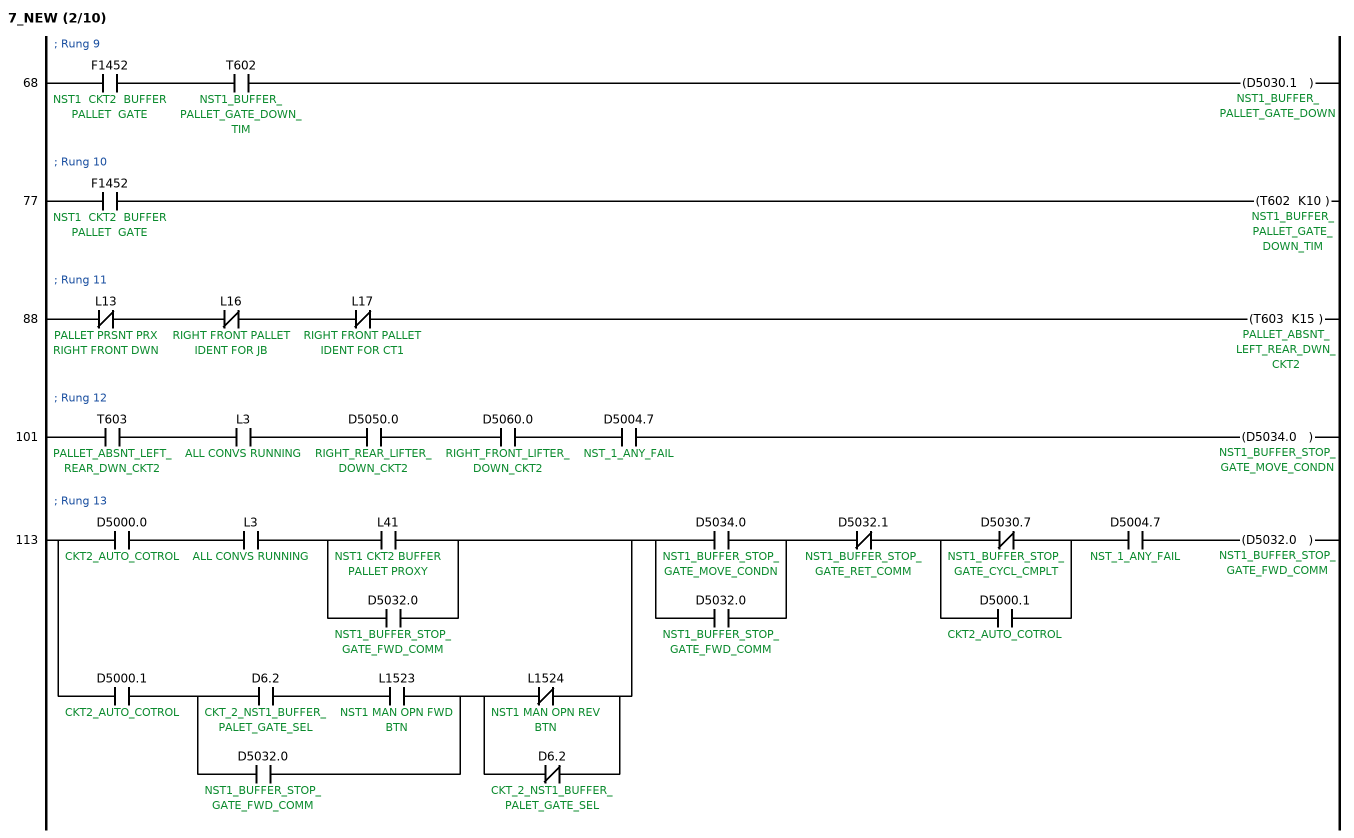
[picture p72: ladder of 7_NEW, rungs at steps 68 to 113]
; Rung 9
68    LD      F1452  ; NST1  CKT2  BUFFER  PALLET  GATE
      AND     T602  ; NST1_BUFFER_PALLET_GATE_DOWN_TIM
      OUT     D5030.1  ; NST1_BUFFER_PALLET_GATE_DOWN
; Rung 10
77    LD      F1452  ; NST1  CKT2  BUFFER  PALLET  GATE
      OUT     T602 K10  ; NST1_BUFFER_PALLET_GATE_DOWN_TIM
; Rung 11
88    LDI     L13  ; PALLET PRSNT PRX RIGHT FRONT DWN
      ANI     L16  ; RIGHT FRONT PALLET IDENT FOR JB
      ANI     L17  ; RIGHT FRONT PALLET IDENT FOR CT1
      OUT     T603 K15  ; PALLET_ABSNT_LEFT_REAR_DWN_CKT2
; Rung 12
101   LD      T603  ; PALLET_ABSNT_LEFT_REAR_DWN_CKT2
      AND     L3  ; ALL CONVS RUNNING
      AND     D5050.0  ; RIGHT_REAR_LIFTER_DOWN_CKT2
      AND     D5060.0  ; RIGHT_FRONT_LIFTER_DOWN_CKT2
      AND     D5004.7  ; NST_1_ANY_FAIL
      OUT     D5034.0  ; NST1_BUFFER_STOP_GATE_MOVE_CONDN
; Rung 13
113   LD      D5000.0  ; CKT2_AUTO_COTROL
      AND     L3  ; ALL CONVS RUNNING
      LD      L41  ; NST1 CKT2 BUFFER PALLET PROXY
      OR      D5032.0  ; NST1_BUFFER_STOP_GATE_FWD_COMM
      ANB
      LD      D5000.1  ; CKT2_AUTO_COTROL
      LD      D6.2  ; CKT_2_NST1_BUFFER_PALET_GATE_SEL
      AND     L1523  ; NST1 MAN OPN FWD BTN
      OR      D5032.0  ; NST1_BUFFER_STOP_GATE_FWD_COMM
      ANB
      LDI     L1524  ; NST1 MAN OPN REV BTN
      ORI     D6.2  ; CKT_2_NST1_BUFFER_PALET_GATE_SEL
      ANB
      ORB
      LD      D5034.0  ; NST1_BUFFER_STOP_GATE_MOVE_CONDN
      OR      D5032.0  ; NST1_BUFFER_STOP_GATE_FWD_COMM
      ANB
      ANI     D5032.1  ; NST1_BUFFER_STOP_GATE_RET_COMM
      LDI     D5030.7  ; NST1_BUFFER_STOP_GATE_CYCL_CMPLT
      OR      D5000.1  ; CKT2_AUTO_COTROL
      ANB
      AND     D5004.7  ; NST_1_ANY_FAIL
      OUT     D5032.0  ; NST1_BUFFER_STOP_GATE_FWD_COMM
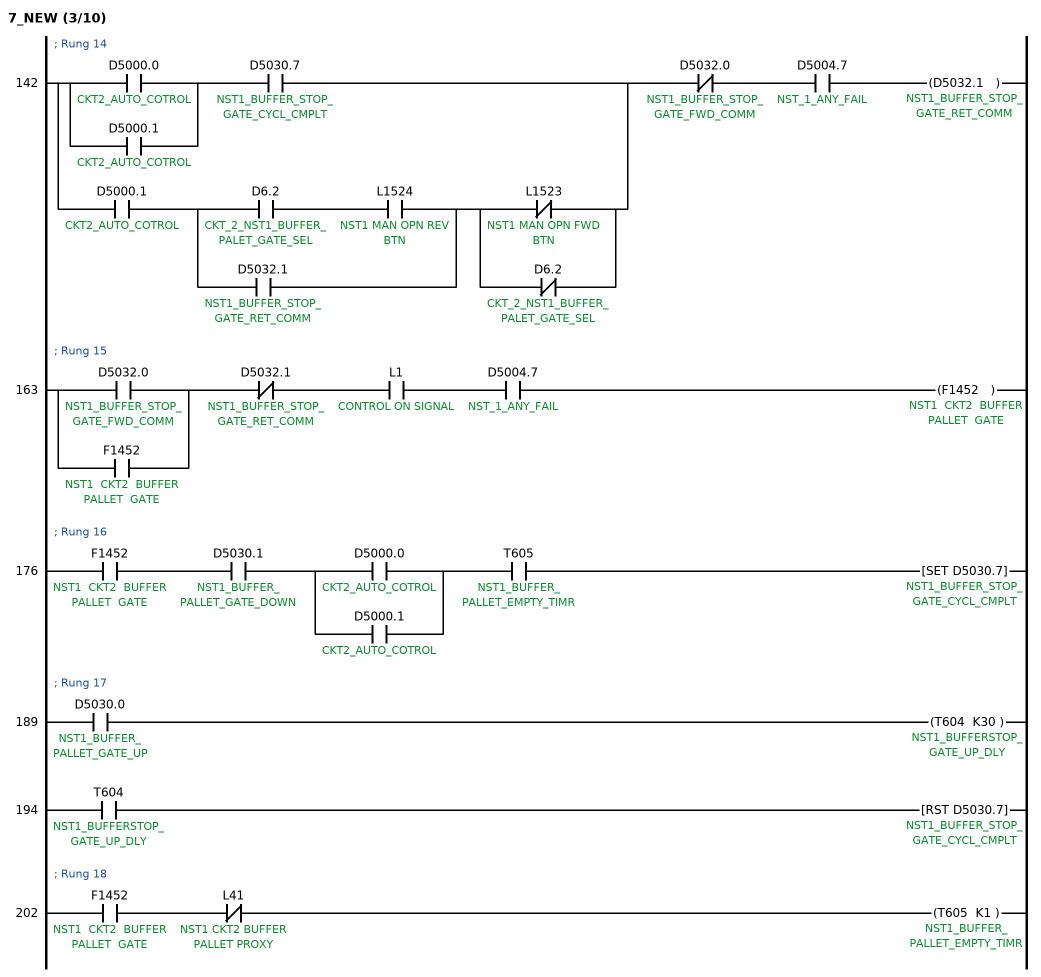
; Rung 14
142   LD      D5000.0  ; CKT2_AUTO_COTROL
      OR      D5000.1  ; CKT2_AUTO_COTROL
      AND     D5030.7  ; NST1_BUFFER_STOP_GATE_CYCL_CMPLT
      LD      D5000.1  ; CKT2_AUTO_COTROL
      LD      D6.2  ; CKT_2_NST1_BUFFER_PALET_GATE_SEL
      AND     L1524  ; NST1 MAN OPN REV BTN
      OR      D5032.1  ; NST1_BUFFER_STOP_GATE_RET_COMM
      ANB
      LDI     L1523  ; NST1 MAN OPN FWD BTN
      ORI     D6.2  ; CKT_2_NST1_BUFFER_PALET_GATE_SEL
      ANB
      ORB
      ANI     D5032.0  ; NST1_BUFFER_STOP_GATE_FWD_COMM
      AND     D5004.7  ; NST_1_ANY_FAIL
      OUT     D5032.1  ; NST1_BUFFER_STOP_GATE_RET_COMM
; Rung 15
163   LD      D5032.0  ; NST1_BUFFER_STOP_GATE_FWD_COMM
      OR      F1452  ; NST1  CKT2  BUFFER  PALLET  GATE
      ANI     D5032.1  ; NST1_BUFFER_STOP_GATE_RET_COMM
      AND     L1  ; CONTROL ON SIGNAL
      AND     D5004.7  ; NST_1_ANY_FAIL
      OUT     F1452  ; NST1  CKT2  BUFFER  PALLET  GATE
; Rung 16
176   LD      F1452  ; NST1  CKT2  BUFFER  PALLET  GATE
      AND     D5030.1  ; NST1_BUFFER_PALLET_GATE_DOWN
      LD      D5000.0  ; CKT2_AUTO_COTROL
      OR      D5000.1  ; CKT2_AUTO_COTROL
      ANB
      AND     T605  ; NST1_BUFFER_PALLET_EMPTY_TIMR
      SET     D5030.7  ; NST1_BUFFER_STOP_GATE_CYCL_CMPLT
; Rung 17
189   LD      D5030.0  ; NST1_BUFFER_PALLET_GATE_UP
      OUT     T604 K30  ; NST1_BUFFERSTOP_GATE_UP_DLY
194   LD      T604  ; NST1_BUFFERSTOP_GATE_UP_DLY
      RST     D5030.7  ; NST1_BUFFER_STOP_GATE_CYCL_CMPLT
; Rung 18
202   LD      F1452  ; NST1  CKT2  BUFFER  PALLET  GATE
      ANI     L41  ; NST1 CKT2 BUFFER PALLET PROXY
      OUT     T605 K1  ; NST1_BUFFER_PALLET_EMPTY_TIMR
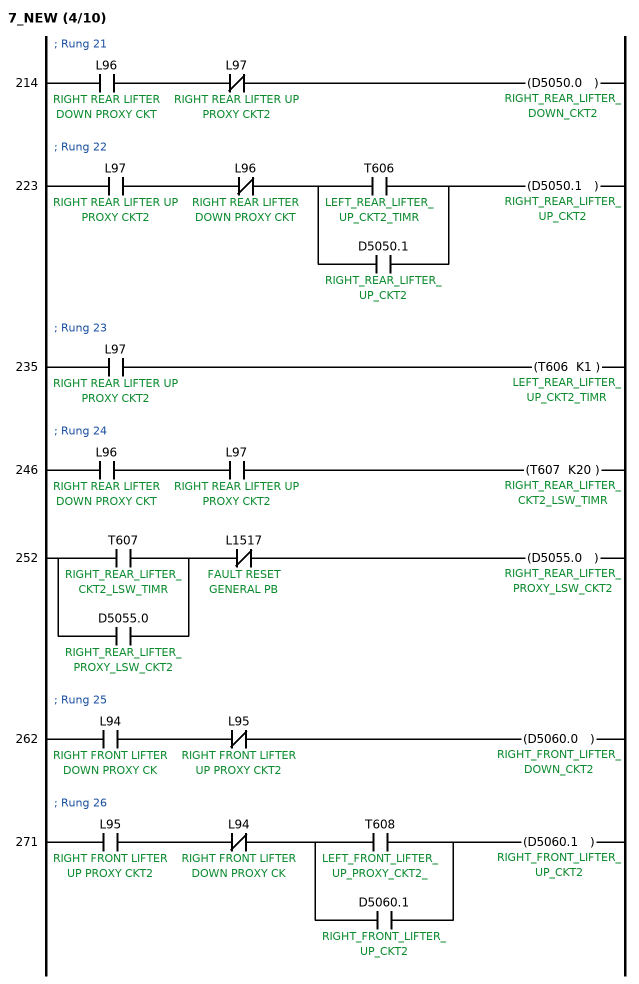
; Rung 21
214   LD      L96  ; RIGHT REAR LIFTER DOWN PROXY CKT
      ANI     L97  ; RIGHT REAR LIFTER UP PROXY CKT2
      OUT     D5050.0  ; RIGHT_REAR_LIFTER_DOWN_CKT2
; Rung 22
223   LD      L97  ; RIGHT REAR LIFTER UP PROXY CKT2
      ANI     L96  ; RIGHT REAR LIFTER DOWN PROXY CKT
      LD      T606  ; LEFT_REAR_LIFTER_UP_CKT2_TIMR
      OR      D5050.1  ; RIGHT_REAR_LIFTER_UP_CKT2
      ANB
      OUT     D5050.1  ; RIGHT_REAR_LIFTER_UP_CKT2
; Rung 23
235   LD      L97  ; RIGHT REAR LIFTER UP PROXY CKT2
      OUT     T606 K1  ; LEFT_REAR_LIFTER_UP_CKT2_TIMR
; Rung 24
246   LD      L96  ; RIGHT REAR LIFTER DOWN PROXY CKT
      AND     L97  ; RIGHT REAR LIFTER UP PROXY CKT2
      OUT     T607 K20  ; RIGHT_REAR_LIFTER_CKT2_LSW_TIMR
252   LD      T607  ; RIGHT_REAR_LIFTER_CKT2_LSW_TIMR
      OR      D5055.0  ; RIGHT_REAR_LIFTER_PROXY_LSW_CKT2
      ANI     L1517  ; FAULT RESET GENERAL PB
      OUT     D5055.0  ; RIGHT_REAR_LIFTER_PROXY_LSW_CKT2
; Rung 25
262   LD      L94  ; RIGHT FRONT LIFTER DOWN PROXY CK
      ANI     L95  ; RIGHT FRONT LIFTER UP PROXY CKT2
      OUT     D5060.0  ; RIGHT_FRONT_LIFTER_DOWN_CKT2
; Rung 26
271   LD      L95  ; RIGHT FRONT LIFTER UP PROXY CKT2
      ANI     L94  ; RIGHT FRONT LIFTER DOWN PROXY CK
      LD      T608  ; LEFT_FRONT_LIFTER_UP_PROXY_CKT2_
      OR      D5060.1  ; RIGHT_FRONT_LIFTER_UP_CKT2
      ANB
      OUT     D5060.1  ; RIGHT_FRONT_LIFTER_UP_CKT2
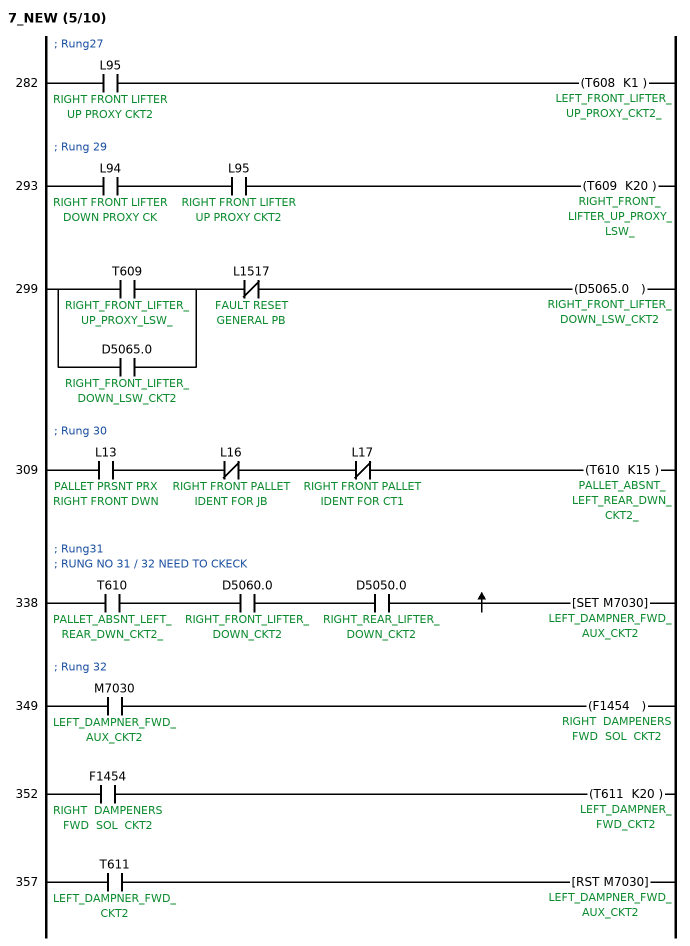
; Rung27
282   LD      L95  ; RIGHT FRONT LIFTER UP PROXY CKT2
      OUT     T608 K1  ; LEFT_FRONT_LIFTER_UP_PROXY_CKT2_
; Rung 29
293   LD      L94  ; RIGHT FRONT LIFTER DOWN PROXY CK
      AND     L95  ; RIGHT FRONT LIFTER UP PROXY CKT2
      OUT     T609 K20  ; RIGHT_FRONT_LIFTER_UP_PROXY_LSW_
299   LD      T609  ; RIGHT_FRONT_LIFTER_UP_PROXY_LSW_
      OR      D5065.0  ; RIGHT_FRONT_LIFTER_DOWN_LSW_CKT2
      ANI     L1517  ; FAULT RESET GENERAL PB
      OUT     D5065.0  ; RIGHT_FRONT_LIFTER_DOWN_LSW_CKT2
; Rung 30
309   LD      L13  ; PALLET PRSNT PRX RIGHT FRONT DWN
      ANI     L16  ; RIGHT FRONT PALLET IDENT FOR JB
      ANI     L17  ; RIGHT FRONT PALLET IDENT FOR CT1
      OUT     T610 K15  ; PALLET_ABSNT_LEFT_REAR_DWN_CKT2_
; Rung31
; RUNG NO 31 / 32 NEED TO CKECK
338   LD      T610  ; PALLET_ABSNT_LEFT_REAR_DWN_CKT2_
      AND     D5060.0  ; RIGHT_FRONT_LIFTER_DOWN_CKT2
      AND     D5050.0  ; RIGHT_REAR_LIFTER_DOWN_CKT2
      MEP
      SET     M7030  ; LEFT_DAMPNER_FWD_AUX_CKT2
; Rung 32
349   LD      M7030  ; LEFT_DAMPNER_FWD_AUX_CKT2
      OUT     F1454  ; RIGHT  DAMPENERS  FWD  SOL  CKT2
352   LD      F1454  ; RIGHT  DAMPENERS  FWD  SOL  CKT2
      OUT     T611 K20  ; LEFT_DAMPNER_FWD_CKT2
357   LD      T611  ; LEFT_DAMPNER_FWD_CKT2
      RST     M7030  ; LEFT_DAMPNER_FWD_AUX_CKT2
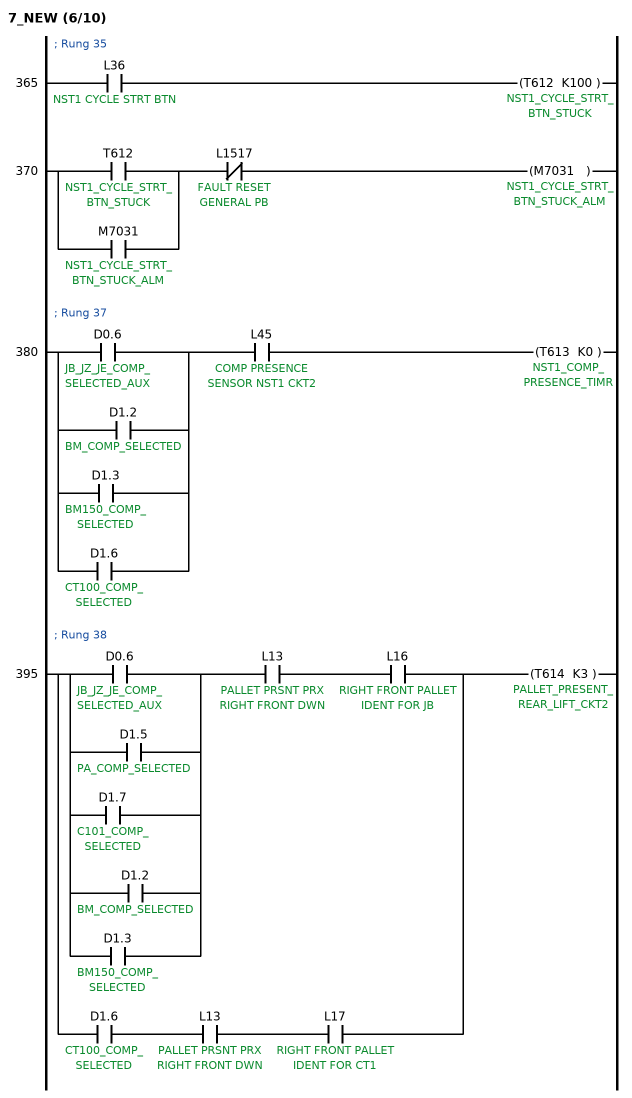
; Rung 35
365   LD      L36  ; NST1 CYCLE STRT BTN
      OUT     T612 K100  ; NST1_CYCLE_STRT_BTN_STUCK
370   LD      T612  ; NST1_CYCLE_STRT_BTN_STUCK
      OR      M7031  ; NST1_CYCLE_STRT_BTN_STUCK_ALM
      ANI     L1517  ; FAULT RESET GENERAL PB
      OUT     M7031  ; NST1_CYCLE_STRT_BTN_STUCK_ALM
; Rung 37
380   LD      D0.6  ; JB_JZ_JE_COMP_SELECTED_AUX
      OR      D1.2  ; BM_COMP_SELECTED
      OR      D1.3  ; BM150_COMP_SELECTED
      OR      D1.6  ; CT100_COMP_SELECTED
      AND     L45  ; COMP PRESENCE SENSOR NST1 CKT2
      OUT     T613 K0  ; NST1_COMP_PRESENCE_TIMR
; Rung 38
395   LD      D0.6  ; JB_JZ_JE_COMP_SELECTED_AUX
      OR      D1.5  ; PA_COMP_SELECTED
      OR      D1.7  ; C101_COMP_SELECTED
      OR      D1.2  ; BM_COMP_SELECTED
      OR      D1.3  ; BM150_COMP_SELECTED
      AND     L13  ; PALLET PRSNT PRX RIGHT FRONT DWN
      AND     L16  ; RIGHT FRONT PALLET IDENT FOR JB
      LD      D1.6  ; CT100_COMP_SELECTED
      AND     L13  ; PALLET PRSNT PRX RIGHT FRONT DWN
      AND     L17  ; RIGHT FRONT PALLET IDENT FOR CT1
      ORB
      OUT     T614 K3  ; PALLET_PRESENT_REAR_LIFT_CKT2
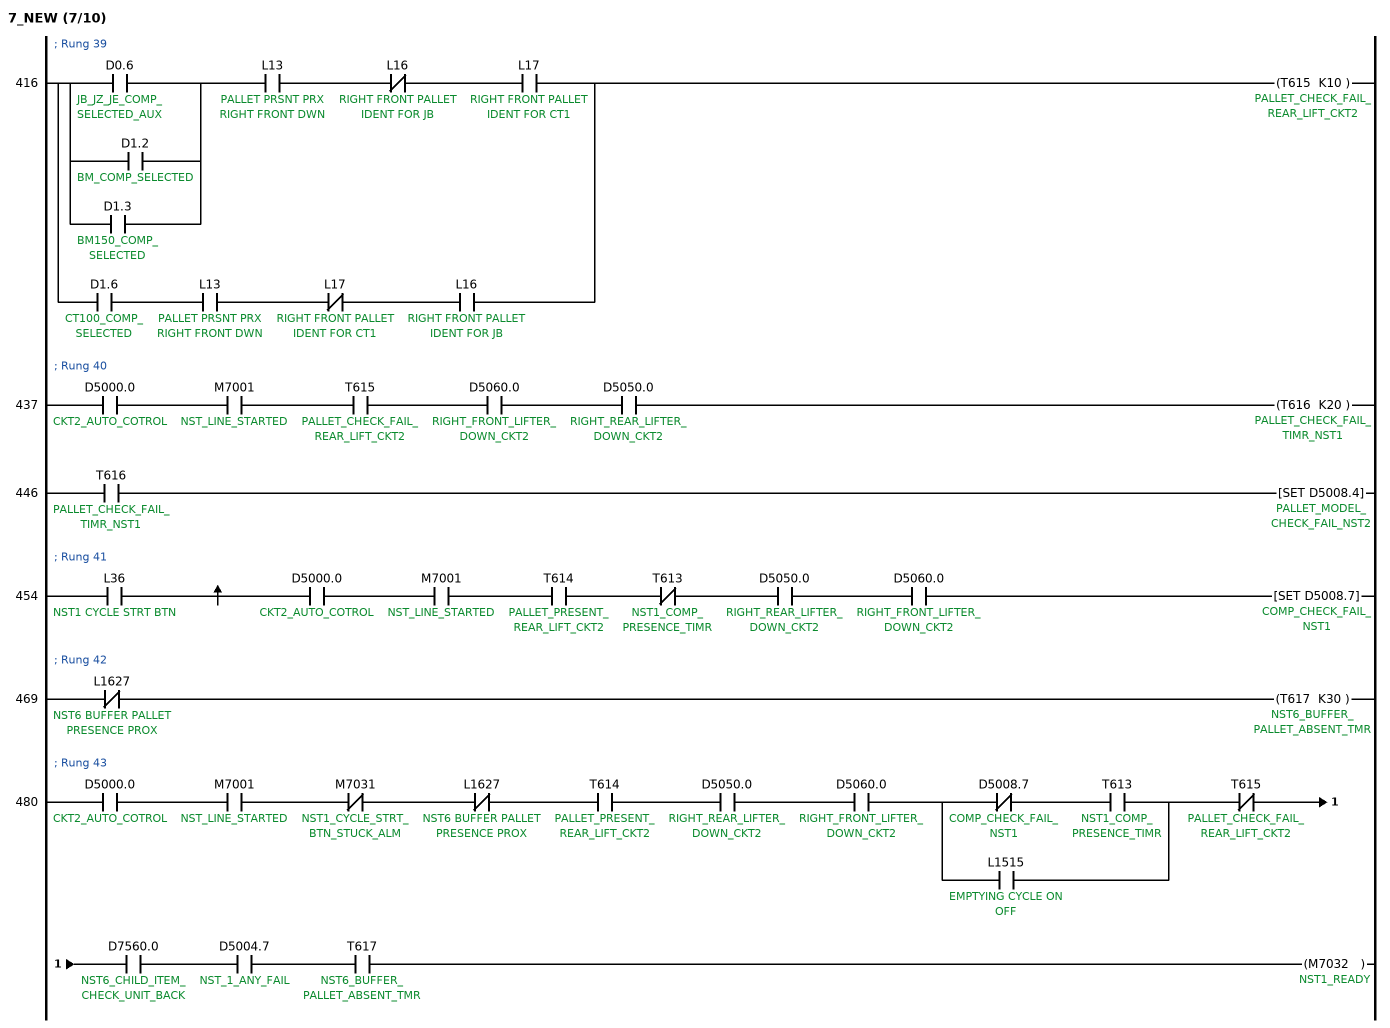
; Rung 39
416   LD      D0.6  ; JB_JZ_JE_COMP_SELECTED_AUX
      OR      D1.2  ; BM_COMP_SELECTED
      OR      D1.3  ; BM150_COMP_SELECTED
      AND     L13  ; PALLET PRSNT PRX RIGHT FRONT DWN
      ANI     L16  ; RIGHT FRONT PALLET IDENT FOR JB
      AND     L17  ; RIGHT FRONT PALLET IDENT FOR CT1
      LD      D1.6  ; CT100_COMP_SELECTED
      AND     L13  ; PALLET PRSNT PRX RIGHT FRONT DWN
      ANI     L17  ; RIGHT FRONT PALLET IDENT FOR CT1
      AND     L16  ; RIGHT FRONT PALLET IDENT FOR JB
      ORB
      OUT     T615 K10  ; PALLET_CHECK_FAIL_REAR_LIFT_CKT2
; Rung 40
437   LD      D5000.0  ; CKT2_AUTO_COTROL
      AND     M7001  ; NST_LINE_STARTED
      AND     T615  ; PALLET_CHECK_FAIL_REAR_LIFT_CKT2
      AND     D5060.0  ; RIGHT_FRONT_LIFTER_DOWN_CKT2
      AND     D5050.0  ; RIGHT_REAR_LIFTER_DOWN_CKT2
      OUT     T616 K20  ; PALLET_CHECK_FAIL_TIMR_NST1
446   LD      T616  ; PALLET_CHECK_FAIL_TIMR_NST1
      SET     D5008.4  ; PALLET_MODEL_CHECK_FAIL_NST2
; Rung 41
454   LD      L36  ; NST1 CYCLE STRT BTN
      MEP
      AND     D5000.0  ; CKT2_AUTO_COTROL
      AND     M7001  ; NST_LINE_STARTED
      AND     T614  ; PALLET_PRESENT_REAR_LIFT_CKT2
      ANI     T613  ; NST1_COMP_PRESENCE_TIMR
      AND     D5050.0  ; RIGHT_REAR_LIFTER_DOWN_CKT2
      AND     D5060.0  ; RIGHT_FRONT_LIFTER_DOWN_CKT2
      SET     D5008.7  ; COMP_CHECK_FAIL_NST1
; Rung 42
469   LDI     L1627  ; NST6 BUFFER PALLET PRESENCE PROX
      OUT     T617 K30  ; NST6_BUFFER_PALLET_ABSENT_TMR
; Rung 43
480   LD      D5000.0  ; CKT2_AUTO_COTROL
      AND     M7001  ; NST_LINE_STARTED
      ANI     M7031  ; NST1_CYCLE_STRT_BTN_STUCK_ALM
      ANI     L1627  ; NST6 BUFFER PALLET PRESENCE PROX
      AND     T614  ; PALLET_PRESENT_REAR_LIFT_CKT2
      AND     D5050.0  ; RIGHT_REAR_LIFTER_DOWN_CKT2
      AND     D5060.0  ; RIGHT_FRONT_LIFTER_DOWN_CKT2
      LDI     D5008.7  ; COMP_CHECK_FAIL_NST1
      AND     T613  ; NST1_COMP_PRESENCE_TIMR
      OR      L1515  ; EMPTYING CYCLE ON OFF
      ANB
      ANI     T615  ; PALLET_CHECK_FAIL_REAR_LIFT_CKT2
      AND     D7560.0  ; NST6_CHILD_ITEM_CHECK_UNIT_BACK
      AND     D5004.7  ; NST_1_ANY_FAIL
      AND     T617  ; NST6_BUFFER_PALLET_ABSENT_TMR
      OUT     M7032  ; NST1_READY
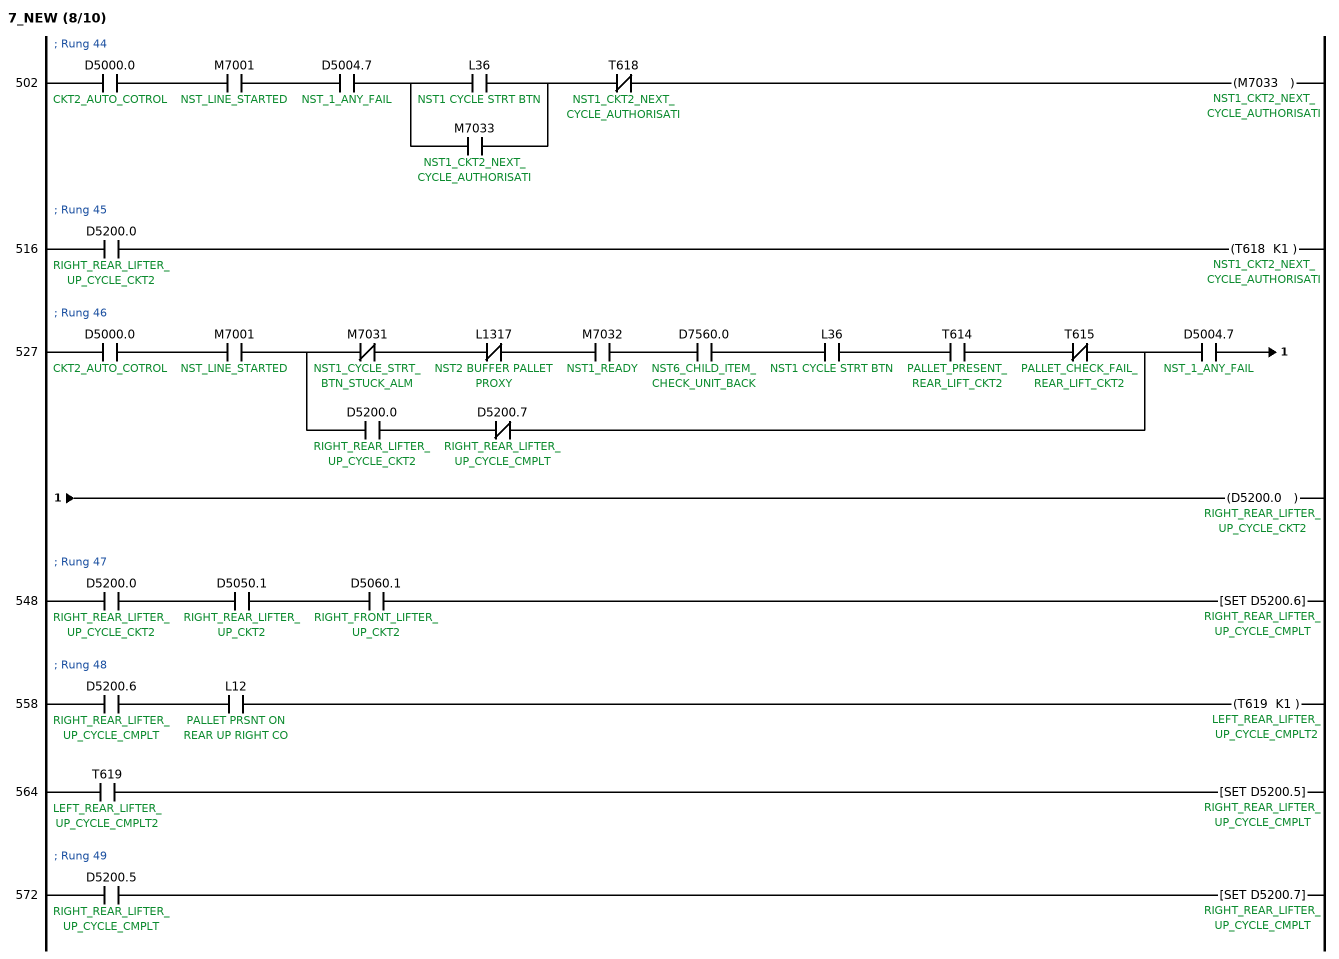
; Rung 44
502   LD      D5000.0  ; CKT2_AUTO_COTROL
      AND     M7001  ; NST_LINE_STARTED
      AND     D5004.7  ; NST_1_ANY_FAIL
      LD      L36  ; NST1 CYCLE STRT BTN
      OR      M7033  ; NST1_CKT2_NEXT_CYCLE_AUTHORISATI
      ANB
      ANI     T618  ; NST1_CKT2_NEXT_CYCLE_AUTHORISATI
      OUT     M7033  ; NST1_CKT2_NEXT_CYCLE_AUTHORISATI
; Rung 45
516   LD      D5200.0  ; RIGHT_REAR_LIFTER_UP_CYCLE_CKT2
      OUT     T618 K1  ; NST1_CKT2_NEXT_CYCLE_AUTHORISATI
; Rung 46
527   LD      D5000.0  ; CKT2_AUTO_COTROL
      AND     M7001  ; NST_LINE_STARTED
      LDI     M7031  ; NST1_CYCLE_STRT_BTN_STUCK_ALM
      ANI     L1317  ; NST2 BUFFER PALLET PROXY
      AND     M7032  ; NST1_READY
      AND     D7560.0  ; NST6_CHILD_ITEM_CHECK_UNIT_BACK
      AND     L36  ; NST1 CYCLE STRT BTN
      AND     T614  ; PALLET_PRESENT_REAR_LIFT_CKT2
      ANI     T615  ; PALLET_CHECK_FAIL_REAR_LIFT_CKT2
      LD      D5200.0  ; RIGHT_REAR_LIFTER_UP_CYCLE_CKT2
      ANI     D5200.7  ; RIGHT_REAR_LIFTER_UP_CYCLE_CMPLT
      ORB
      ANB
      AND     D5004.7  ; NST_1_ANY_FAIL
      OUT     D5200.0  ; RIGHT_REAR_LIFTER_UP_CYCLE_CKT2
; Rung 47
548   LD      D5200.0  ; RIGHT_REAR_LIFTER_UP_CYCLE_CKT2
      AND     D5050.1  ; RIGHT_REAR_LIFTER_UP_CKT2
      AND     D5060.1  ; RIGHT_FRONT_LIFTER_UP_CKT2
      SET     D5200.6  ; RIGHT_REAR_LIFTER_UP_CYCLE_CMPLT
; Rung 48
558   LD      D5200.6  ; RIGHT_REAR_LIFTER_UP_CYCLE_CMPLT
      AND     L12  ; PALLET PRSNT ON REAR UP RIGHT CO
      OUT     T619 K1  ; LEFT_REAR_LIFTER_UP_CYCLE_CMPLT2
564   LD      T619  ; LEFT_REAR_LIFTER_UP_CYCLE_CMPLT2
      SET     D5200.5  ; RIGHT_REAR_LIFTER_UP_CYCLE_CMPLT
; Rung 49
572   LD      D5200.5  ; RIGHT_REAR_LIFTER_UP_CYCLE_CMPLT
      SET     D5200.7  ; RIGHT_REAR_LIFTER_UP_CYCLE_CMPLT
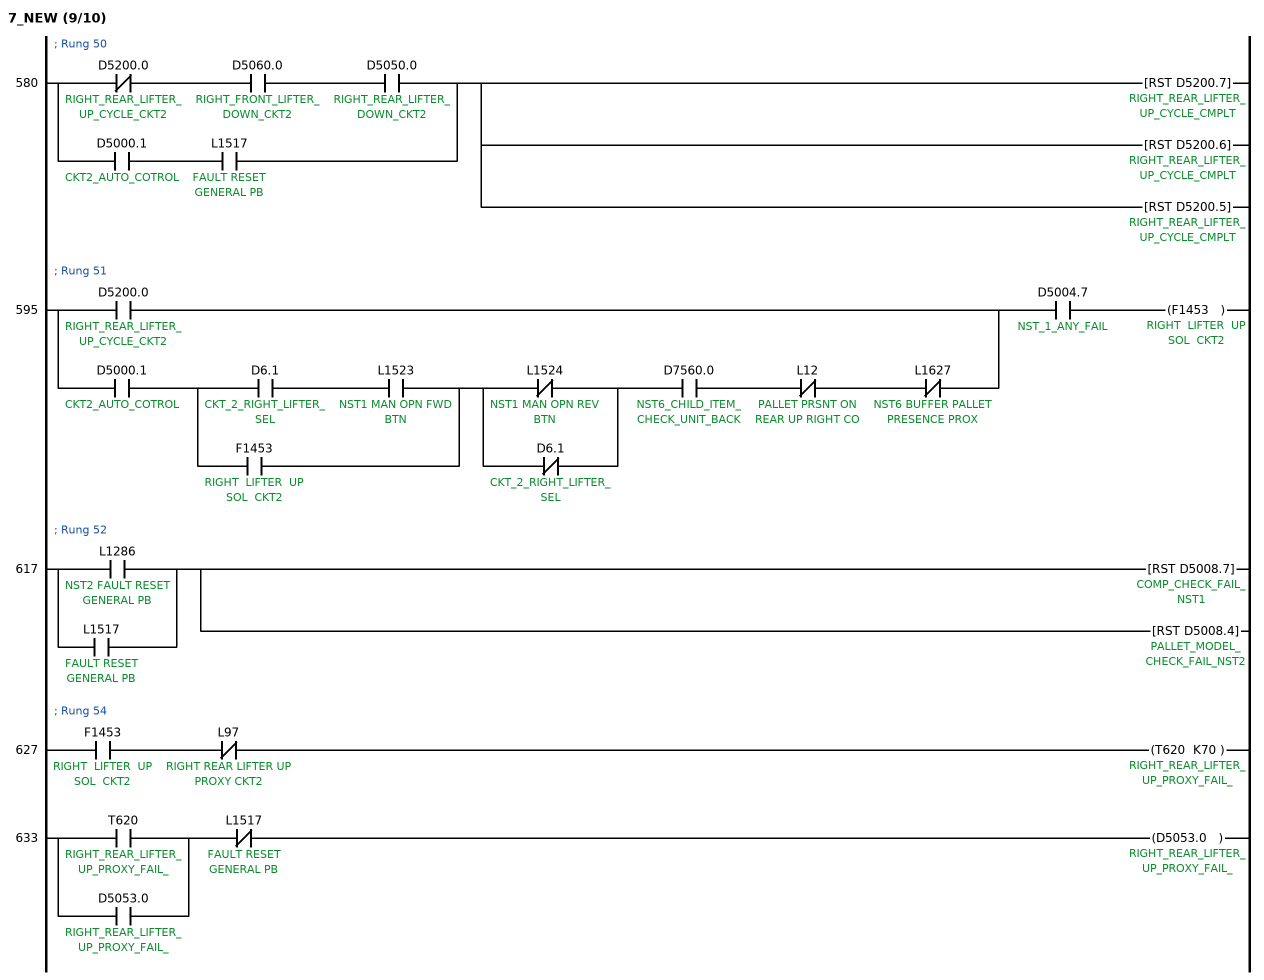
; Rung 50
580   LDI     D5200.0  ; RIGHT_REAR_LIFTER_UP_CYCLE_CKT2
      AND     D5060.0  ; RIGHT_FRONT_LIFTER_DOWN_CKT2
      AND     D5050.0  ; RIGHT_REAR_LIFTER_DOWN_CKT2
      LD      D5000.1  ; CKT2_AUTO_COTROL
      AND     L1517  ; FAULT RESET GENERAL PB
      ORB
      RST     D5200.7  ; RIGHT_REAR_LIFTER_UP_CYCLE_CMPLT
      RST     D5200.6  ; RIGHT_REAR_LIFTER_UP_CYCLE_CMPLT
      RST     D5200.5  ; RIGHT_REAR_LIFTER_UP_CYCLE_CMPLT
; Rung 51
595   LD      D5200.0  ; RIGHT_REAR_LIFTER_UP_CYCLE_CKT2
      LD      D5000.1  ; CKT2_AUTO_COTROL
      LD      D6.1  ; CKT_2_RIGHT_LIFTER_SEL
      AND     L1523  ; NST1 MAN OPN FWD BTN
      OR      F1453  ; RIGHT  LIFTER  UP  SOL  CKT2
      ANB
      LDI     L1524  ; NST1 MAN OPN REV BTN
      ORI     D6.1  ; CKT_2_RIGHT_LIFTER_SEL
      ANB
      AND     D7560.0  ; NST6_CHILD_ITEM_CHECK_UNIT_BACK
      ANI     L12  ; PALLET PRSNT ON REAR UP RIGHT CO
      ANI     L1627  ; NST6 BUFFER PALLET PRESENCE PROX
      ORB
      AND     D5004.7  ; NST_1_ANY_FAIL
      OUT     F1453  ; RIGHT  LIFTER  UP  SOL  CKT2
; Rung 52
617   LD      L1286  ; NST2 FAULT RESET GENERAL PB
      OR      L1517  ; FAULT RESET GENERAL PB
      RST     D5008.7  ; COMP_CHECK_FAIL_NST1
      RST     D5008.4  ; PALLET_MODEL_CHECK_FAIL_NST2
; Rung 54
627   LD      F1453  ; RIGHT  LIFTER  UP  SOL  CKT2
      ANI     L97  ; RIGHT REAR LIFTER UP PROXY CKT2
      OUT     T620 K70  ; RIGHT_REAR_LIFTER_UP_PROXY_FAIL_
633   LD      T620  ; RIGHT_REAR_LIFTER_UP_PROXY_FAIL_
      OR      D5053.0  ; RIGHT_REAR_LIFTER_UP_PROXY_FAIL_
      ANI     L1517  ; FAULT RESET GENERAL PB
      OUT     D5053.0  ; RIGHT_REAR_LIFTER_UP_PROXY_FAIL_
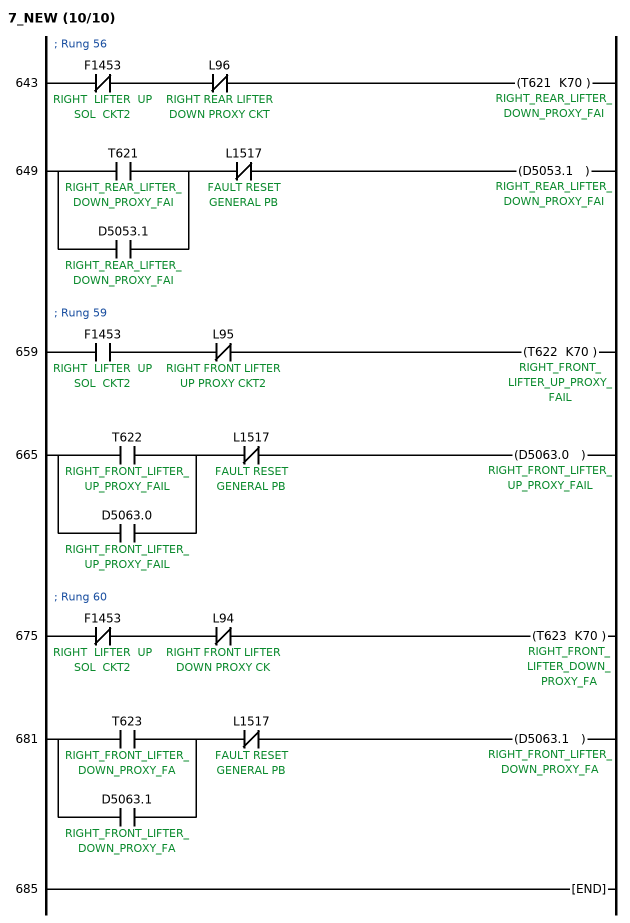
; Rung 56
643   LDI     F1453  ; RIGHT  LIFTER  UP  SOL  CKT2
      ANI     L96  ; RIGHT REAR LIFTER DOWN PROXY CKT
      OUT     T621 K70  ; RIGHT_REAR_LIFTER_DOWN_PROXY_FAI
649   LD      T621  ; RIGHT_REAR_LIFTER_DOWN_PROXY_FAI
      OR      D5053.1  ; RIGHT_REAR_LIFTER_DOWN_PROXY_FAI
      ANI     L1517  ; FAULT RESET GENERAL PB
      OUT     D5053.1  ; RIGHT_REAR_LIFTER_DOWN_PROXY_FAI
; Rung 59
659   LD      F1453  ; RIGHT  LIFTER  UP  SOL  CKT2
      ANI     L95  ; RIGHT FRONT LIFTER UP PROXY CKT2
      OUT     T622 K70  ; RIGHT_FRONT_LIFTER_UP_PROXY_FAIL
665   LD      T622  ; RIGHT_FRONT_LIFTER_UP_PROXY_FAIL
      OR      D5063.0  ; RIGHT_FRONT_LIFTER_UP_PROXY_FAIL
      ANI     L1517  ; FAULT RESET GENERAL PB
      OUT     D5063.0  ; RIGHT_FRONT_LIFTER_UP_PROXY_FAIL
; Rung 60
675   LDI     F1453  ; RIGHT  LIFTER  UP  SOL  CKT2
      ANI     L94  ; RIGHT FRONT LIFTER DOWN PROXY CK
      OUT     T623 K70  ; RIGHT_FRONT_LIFTER_DOWN_PROXY_FA
681   LD      T623  ; RIGHT_FRONT_LIFTER_DOWN_PROXY_FA
      OR      D5063.1  ; RIGHT_FRONT_LIFTER_DOWN_PROXY_FA
      ANI     L1517  ; FAULT RESET GENERAL PB
      OUT     D5063.1  ; RIGHT_FRONT_LIFTER_DOWN_PROXY_FA
685   END
END_PROGRAM

PROGRAM 8_NEW  // ST2 CK2
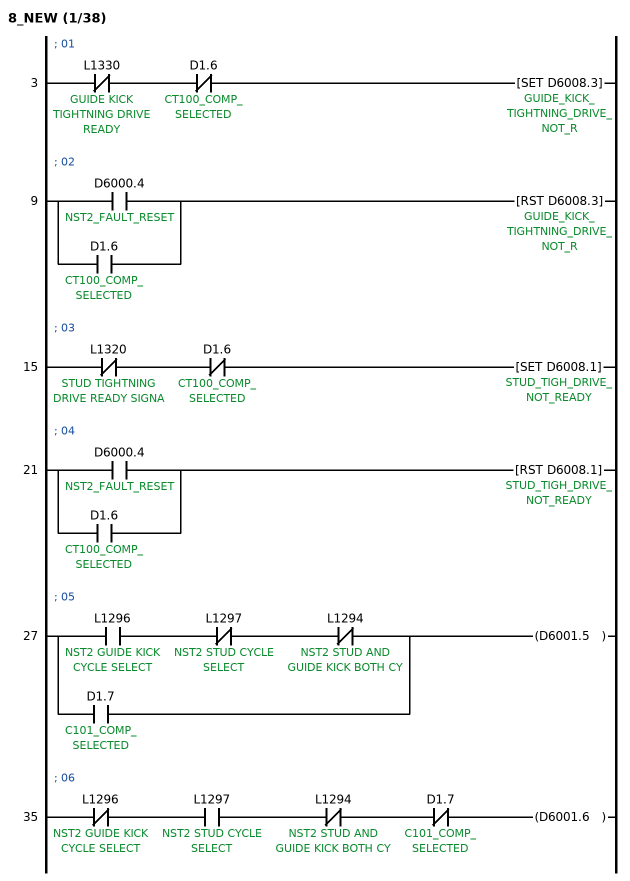
; 01
3     LDI     L1330  ; GUIDE KICK TIGHTNING DRIVE READY
      ANI     D1.6  ; CT100_COMP_SELECTED
      SET     D6008.3  ; GUIDE_KICK_TIGHTNING_DRIVE_NOT_R
; 02
9     LD      D6000.4  ; NST2_FAULT_RESET
      OR      D1.6  ; CT100_COMP_SELECTED
      RST     D6008.3  ; GUIDE_KICK_TIGHTNING_DRIVE_NOT_R
; 03
15    LDI     L1320  ; STUD TIGHTNING DRIVE READY SIGNA
      ANI     D1.6  ; CT100_COMP_SELECTED
      SET     D6008.1  ; STUD_TIGH_DRIVE_NOT_READY
; 04
21    LD      D6000.4  ; NST2_FAULT_RESET
      OR      D1.6  ; CT100_COMP_SELECTED
      RST     D6008.1  ; STUD_TIGH_DRIVE_NOT_READY
; 05
27    LD      L1296  ; NST2 GUIDE KICK CYCLE SELECT
      ANI     L1297  ; NST2 STUD CYCLE SELECT
      ANI     L1294  ; NST2 STUD AND GUIDE KICK BOTH CY
      OR      D1.7  ; C101_COMP_SELECTED
      OUT     D6001.5
; 06
35    LDI     L1296  ; NST2 GUIDE KICK CYCLE SELECT
      AND     L1297  ; NST2 STUD CYCLE SELECT
      ANI     L1294  ; NST2 STUD AND GUIDE KICK BOTH CY
      ANI     D1.7  ; C101_COMP_SELECTED
      OUT     D6001.6
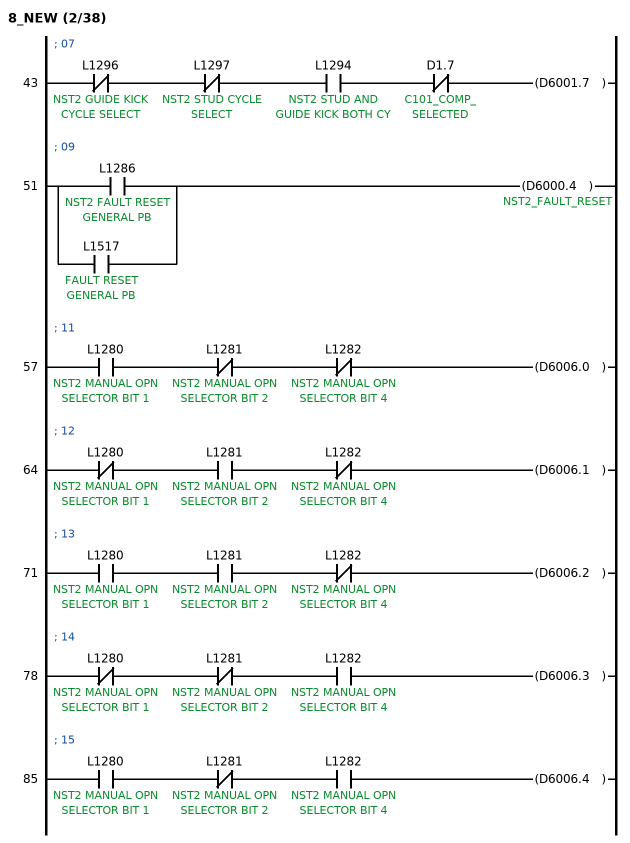
; 07
43    LDI     L1296  ; NST2 GUIDE KICK CYCLE SELECT
      ANI     L1297  ; NST2 STUD CYCLE SELECT
      AND     L1294  ; NST2 STUD AND GUIDE KICK BOTH CY
      ANI     D1.7  ; C101_COMP_SELECTED
      OUT     D6001.7
; 09
51    LD      L1286  ; NST2 FAULT RESET GENERAL PB
      OR      L1517  ; FAULT RESET GENERAL PB
      OUT     D6000.4  ; NST2_FAULT_RESET
; 11
57    LD      L1280  ; NST2 MANUAL OPN SELECTOR BIT 1
      ANI     L1281  ; NST2 MANUAL OPN SELECTOR BIT 2
      ANI     L1282  ; NST2 MANUAL OPN SELECTOR BIT 4
      OUT     D6006.0
; 12
64    LDI     L1280  ; NST2 MANUAL OPN SELECTOR BIT 1
      AND     L1281  ; NST2 MANUAL OPN SELECTOR BIT 2
      ANI     L1282  ; NST2 MANUAL OPN SELECTOR BIT 4
      OUT     D6006.1
; 13
71    LD      L1280  ; NST2 MANUAL OPN SELECTOR BIT 1
      AND     L1281  ; NST2 MANUAL OPN SELECTOR BIT 2
      ANI     L1282  ; NST2 MANUAL OPN SELECTOR BIT 4
      OUT     D6006.2
; 14
78    LDI     L1280  ; NST2 MANUAL OPN SELECTOR BIT 1
      ANI     L1281  ; NST2 MANUAL OPN SELECTOR BIT 2
      AND     L1282  ; NST2 MANUAL OPN SELECTOR BIT 4
      OUT     D6006.3
; 15
85    LD      L1280  ; NST2 MANUAL OPN SELECTOR BIT 1
      ANI     L1281  ; NST2 MANUAL OPN SELECTOR BIT 2
      AND     L1282  ; NST2 MANUAL OPN SELECTOR BIT 4
      OUT     D6006.4
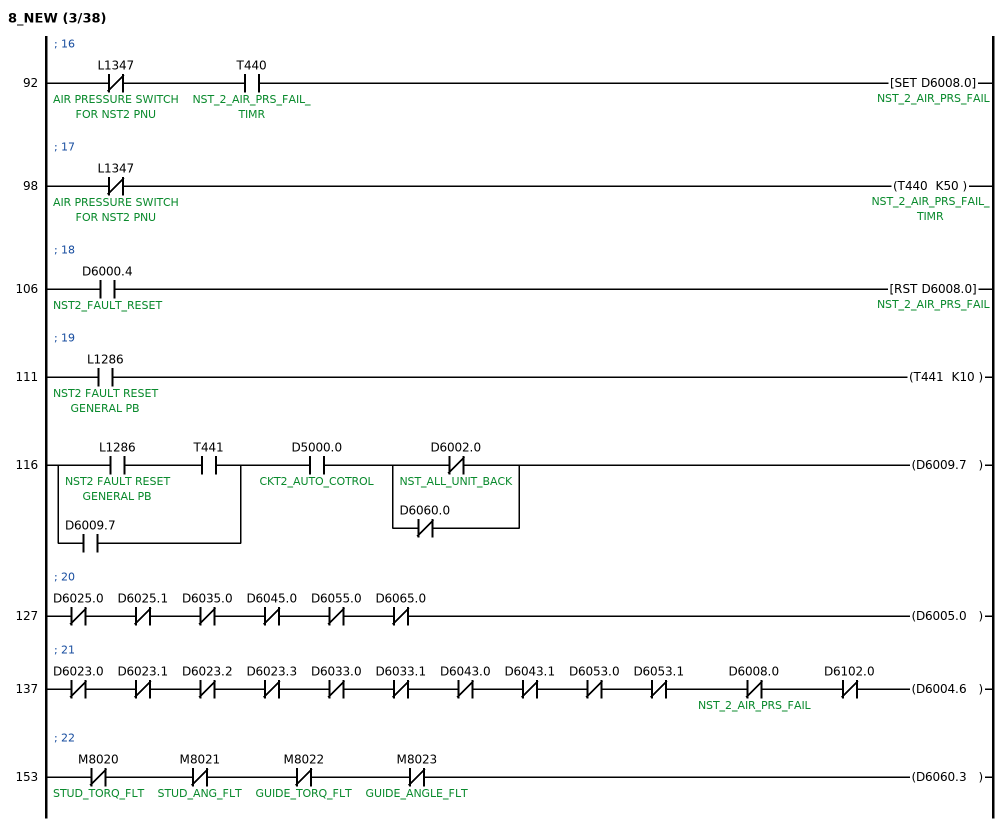
; 16
92    LDI     L1347  ; AIR PRESSURE SWITCH FOR NST2 PNU
      AND     T440  ; NST_2_AIR_PRS_FAIL_TIMR
      SET     D6008.0  ; NST_2_AIR_PRS_FAIL
; 17
98    LDI     L1347  ; AIR PRESSURE SWITCH FOR NST2 PNU
      OUT     T440 K50  ; NST_2_AIR_PRS_FAIL_TIMR
; 18
106   LD      D6000.4  ; NST2_FAULT_RESET
      RST     D6008.0  ; NST_2_AIR_PRS_FAIL
; 19
111   LD      L1286  ; NST2 FAULT RESET GENERAL PB
      OUT     T441 K10
116   LD      L1286  ; NST2 FAULT RESET GENERAL PB
      AND     T441
      OR      D6009.7
      AND     D5000.0  ; CKT2_AUTO_COTROL
      LDI     D6002.0  ; NST_ALL_UNIT_BACK
      ORI     D6060.0
      ANB
      OUT     D6009.7
; 20
127   LDI     D6025.0
      ANI     D6025.1
      ANI     D6035.0
      ANI     D6045.0
      ANI     D6055.0
      ANI     D6065.0
      OUT     D6005.0
; 21
137   LDI     D6023.0
      ANI     D6023.1
      ANI     D6023.2
      ANI     D6023.3
      ANI     D6033.0
      ANI     D6033.1
      ANI     D6043.0
      ANI     D6043.1
      ANI     D6053.0
      ANI     D6053.1
      ANI     D6008.0  ; NST_2_AIR_PRS_FAIL
      ANI     D6102.0
      OUT     D6004.6
; 22
153   LDI     M8020  ; STUD_TORQ_FLT
      ANI     M8021  ; STUD_ANG_FLT
      ANI     M8022  ; GUIDE_TORQ_FLT
      ANI     M8023  ; GUIDE_ANGLE_FLT
      OUT     D6060.3
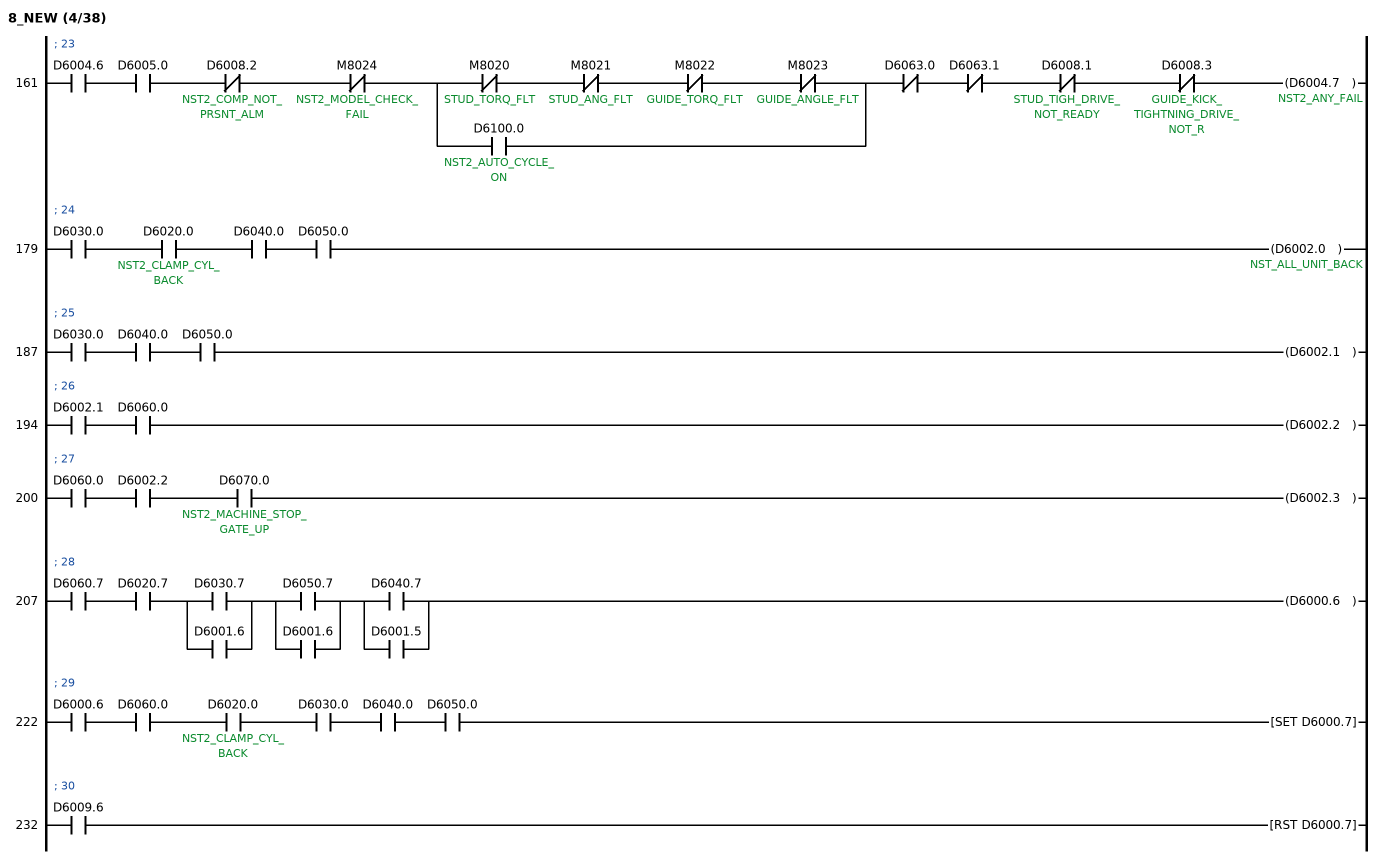
; 23
161   LD      D6004.6
      AND     D6005.0
      ANI     D6008.2  ; NST2_COMP_NOT_PRSNT_ALM
      ANI     M8024  ; NST2_MODEL_CHECK_FAIL
      LDI     M8020  ; STUD_TORQ_FLT
      ANI     M8021  ; STUD_ANG_FLT
      ANI     M8022  ; GUIDE_TORQ_FLT
      ANI     M8023  ; GUIDE_ANGLE_FLT
      OR      D6100.0  ; NST2_AUTO_CYCLE_ON
      ANB
      ANI     D6063.0
      ANI     D6063.1
      ANI     D6008.1  ; STUD_TIGH_DRIVE_NOT_READY
      ANI     D6008.3  ; GUIDE_KICK_TIGHTNING_DRIVE_NOT_R
      OUT     D6004.7  ; NST2_ANY_FAIL
; 24
179   LD      D6030.0
      AND     D6020.0  ; NST2_CLAMP_CYL_BACK
      AND     D6040.0
      AND     D6050.0
      OUT     D6002.0  ; NST_ALL_UNIT_BACK
; 25
187   LD      D6030.0
      AND     D6040.0
      AND     D6050.0
      OUT     D6002.1
; 26
194   LD      D6002.1
      AND     D6060.0
      OUT     D6002.2
; 27
200   LD      D6060.0
      AND     D6002.2
      AND     D6070.0  ; NST2_MACHINE_STOP_GATE_UP
      OUT     D6002.3
; 28
207   LD      D6060.7
      AND     D6020.7
      LD      D6030.7
      OR      D6001.6
      ANB
      LD      D6050.7
      OR      D6001.6
      ANB
      LD      D6040.7
      OR      D6001.5
      ANB
      OUT     D6000.6
; 29
222   LD      D6000.6
      AND     D6060.0
      AND     D6020.0  ; NST2_CLAMP_CYL_BACK
      AND     D6030.0
      AND     D6040.0
      AND     D6050.0
      SET     D6000.7
; 30
232   LD      D6009.6
      RST     D6000.7
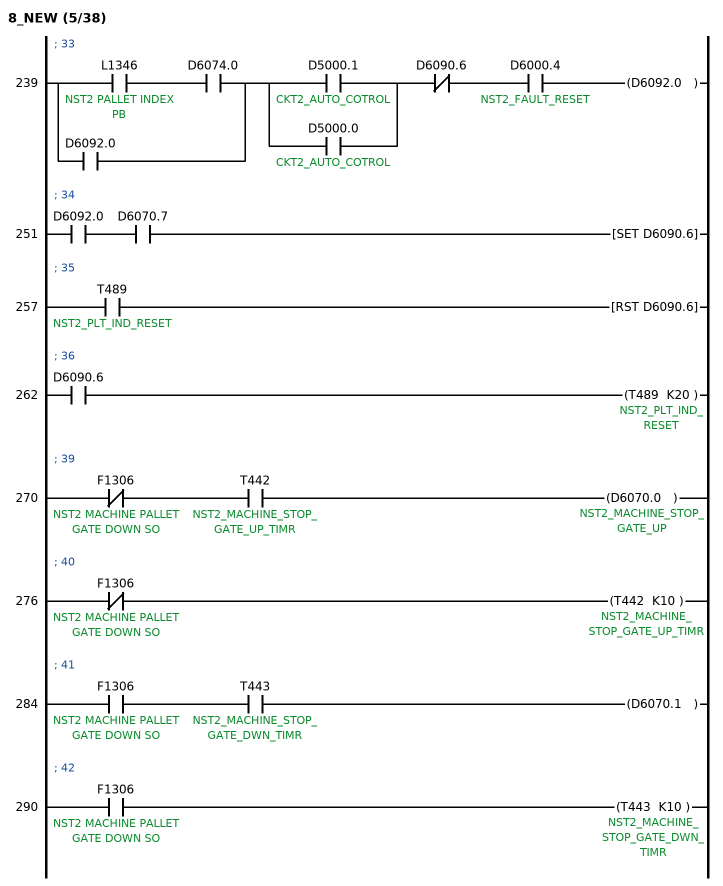
; 
; 33
239   LD      L1346  ; NST2 PALLET INDEX PB
      AND     D6074.0
      OR      D6092.0
      LD      D5000.1  ; CKT2_AUTO_COTROL
      OR      D5000.0  ; CKT2_AUTO_COTROL
      ANB
      ANI     D6090.6
      AND     D6000.4  ; NST2_FAULT_RESET
      OUT     D6092.0
; 34
251   LD      D6092.0
      AND     D6070.7
      SET     D6090.6
; 35
257   LD      T489  ; NST2_PLT_IND_RESET
      RST     D6090.6
; 36
262   LD      D6090.6
      OUT     T489 K20  ; NST2_PLT_IND_RESET
; 39
270   LDI     F1306  ; NST2 MACHINE PALLET GATE DOWN SO
      AND     T442  ; NST2_MACHINE_STOP_GATE_UP_TIMR
      OUT     D6070.0  ; NST2_MACHINE_STOP_GATE_UP
; 40
276   LDI     F1306  ; NST2 MACHINE PALLET GATE DOWN SO
      OUT     T442 K10  ; NST2_MACHINE_STOP_GATE_UP_TIMR
; 41
284   LD      F1306  ; NST2 MACHINE PALLET GATE DOWN SO
      AND     T443  ; NST2_MACHINE_STOP_GATE_DWN_TIMR
      OUT     D6070.1
; 42
290   LD      F1306  ; NST2 MACHINE PALLET GATE DOWN SO
      OUT     T443 K10  ; NST2_MACHINE_STOP_GATE_DWN_TIMR
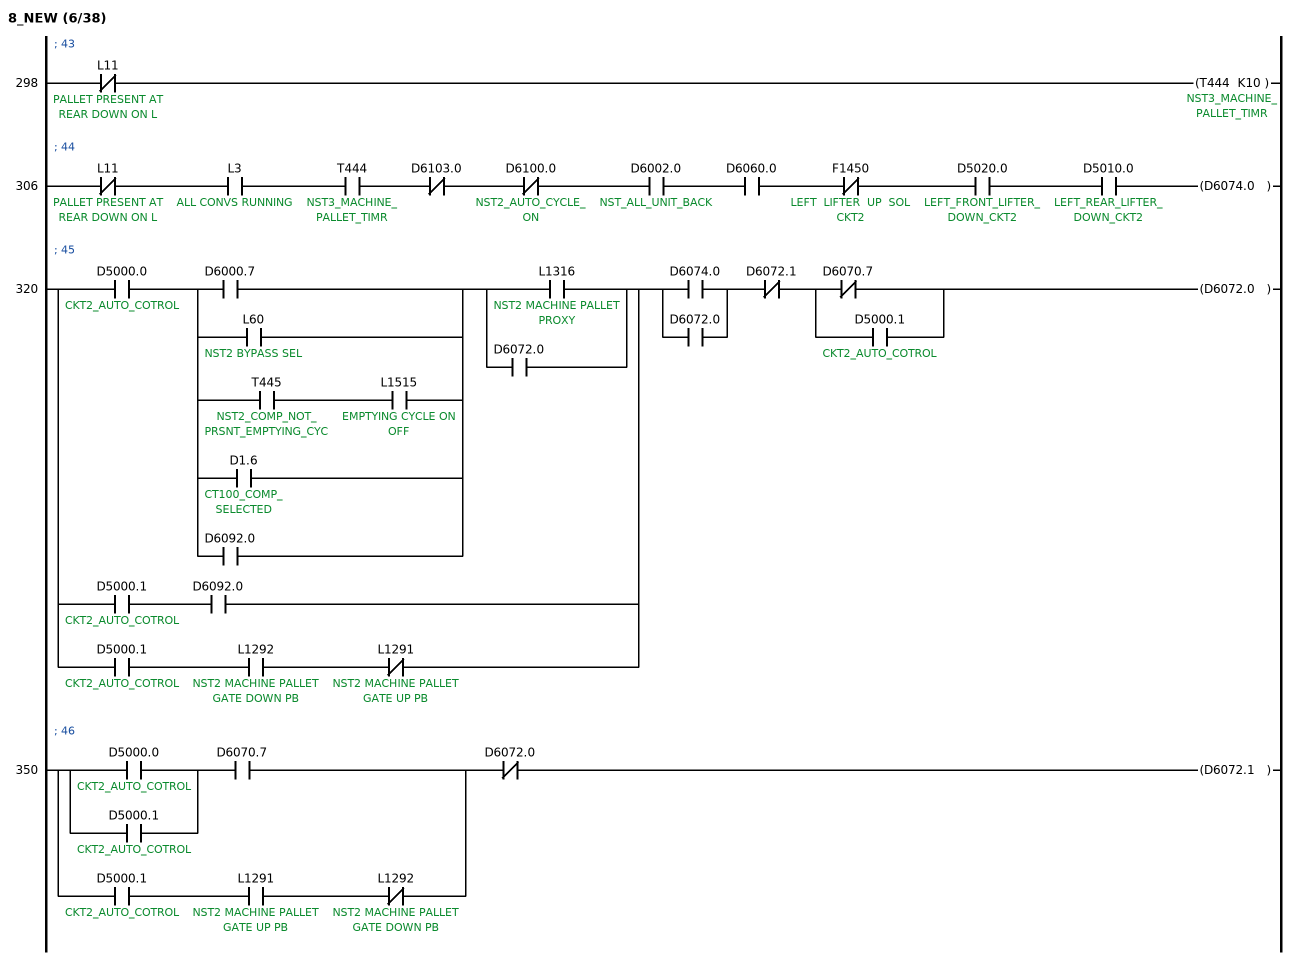
; 43
298   LDI     L11  ; PALLET PRESENT AT REAR DOWN ON L
      OUT     T444 K10  ; NST3_MACHINE_PALLET_TIMR
; 44
306   LDI     L11  ; PALLET PRESENT AT REAR DOWN ON L
      AND     L3  ; ALL CONVS RUNNING
      AND     T444  ; NST3_MACHINE_PALLET_TIMR
      ANI     D6103.0
      ANI     D6100.0  ; NST2_AUTO_CYCLE_ON
      AND     D6002.0  ; NST_ALL_UNIT_BACK
      AND     D6060.0
      ANI     F1450  ; LEFT  LIFTER  UP  SOL  CKT2
      AND     D5020.0  ; LEFT_FRONT_LIFTER_DOWN_CKT2
      AND     D5010.0  ; LEFT_REAR_LIFTER_DOWN_CKT2
      OUT     D6074.0
; 45
320   LD      D5000.0  ; CKT2_AUTO_COTROL
      LD      D6000.7
      OR      L60  ; NST2 BYPASS SEL
      LD      T445  ; NST2_COMP_NOT_PRSNT_EMPTYING_CYC
      AND     L1515  ; EMPTYING CYCLE ON OFF
      ORB
      OR      D1.6  ; CT100_COMP_SELECTED
      OR      D6092.0
      ANB
      LD      L1316  ; NST2 MACHINE PALLET PROXY
      OR      D6072.0
      ANB
      LD      D5000.1  ; CKT2_AUTO_COTROL
      AND     D6092.0
      ORB
      LD      D5000.1  ; CKT2_AUTO_COTROL
      AND     L1292  ; NST2 MACHINE PALLET GATE DOWN PB
      ANI     L1291  ; NST2 MACHINE PALLET GATE UP PB
      ORB
      LD      D6074.0
      OR      D6072.0
      ANB
      ANI     D6072.1
      LDI     D6070.7
      OR      D5000.1  ; CKT2_AUTO_COTROL
      ANB
      OUT     D6072.0
; 46
350   LD      D5000.0  ; CKT2_AUTO_COTROL
      OR      D5000.1  ; CKT2_AUTO_COTROL
      AND     D6070.7
      LD      D5000.1  ; CKT2_AUTO_COTROL
      AND     L1291  ; NST2 MACHINE PALLET GATE UP PB
      ANI     L1292  ; NST2 MACHINE PALLET GATE DOWN PB
      ORB
      ANI     D6072.0
      OUT     D6072.1
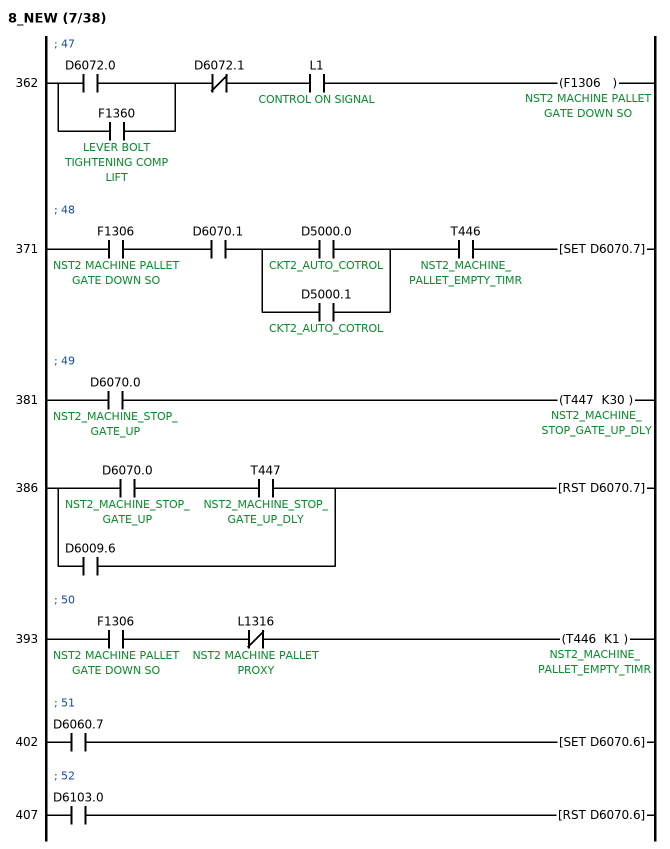
; 47
362   LD      D6072.0
      OR      F1360  ; LEVER BOLT TIGHTENING COMP LIFT
      ANI     D6072.1
      AND     L1  ; CONTROL ON SIGNAL
      OUT     F1306  ; NST2 MACHINE PALLET GATE DOWN SO
; 48
371   LD      F1306  ; NST2 MACHINE PALLET GATE DOWN SO
      AND     D6070.1
      LD      D5000.0  ; CKT2_AUTO_COTROL
      OR      D5000.1  ; CKT2_AUTO_COTROL
      ANB
      AND     T446  ; NST2_MACHINE_PALLET_EMPTY_TIMR
      SET     D6070.7
; 49
381   LD      D6070.0  ; NST2_MACHINE_STOP_GATE_UP
      OUT     T447 K30  ; NST2_MACHINE_STOP_GATE_UP_DLY
386   LD      D6070.0  ; NST2_MACHINE_STOP_GATE_UP
      AND     T447  ; NST2_MACHINE_STOP_GATE_UP_DLY
      OR      D6009.6
      RST     D6070.7
; 50
393   LD      F1306  ; NST2 MACHINE PALLET GATE DOWN SO
      ANI     L1316  ; NST2 MACHINE PALLET PROXY
      OUT     T446 K1  ; NST2_MACHINE_PALLET_EMPTY_TIMR
; 51
402   LD      D6060.7
      SET     D6070.6
; 52
407   LD      D6103.0
      RST     D6070.6
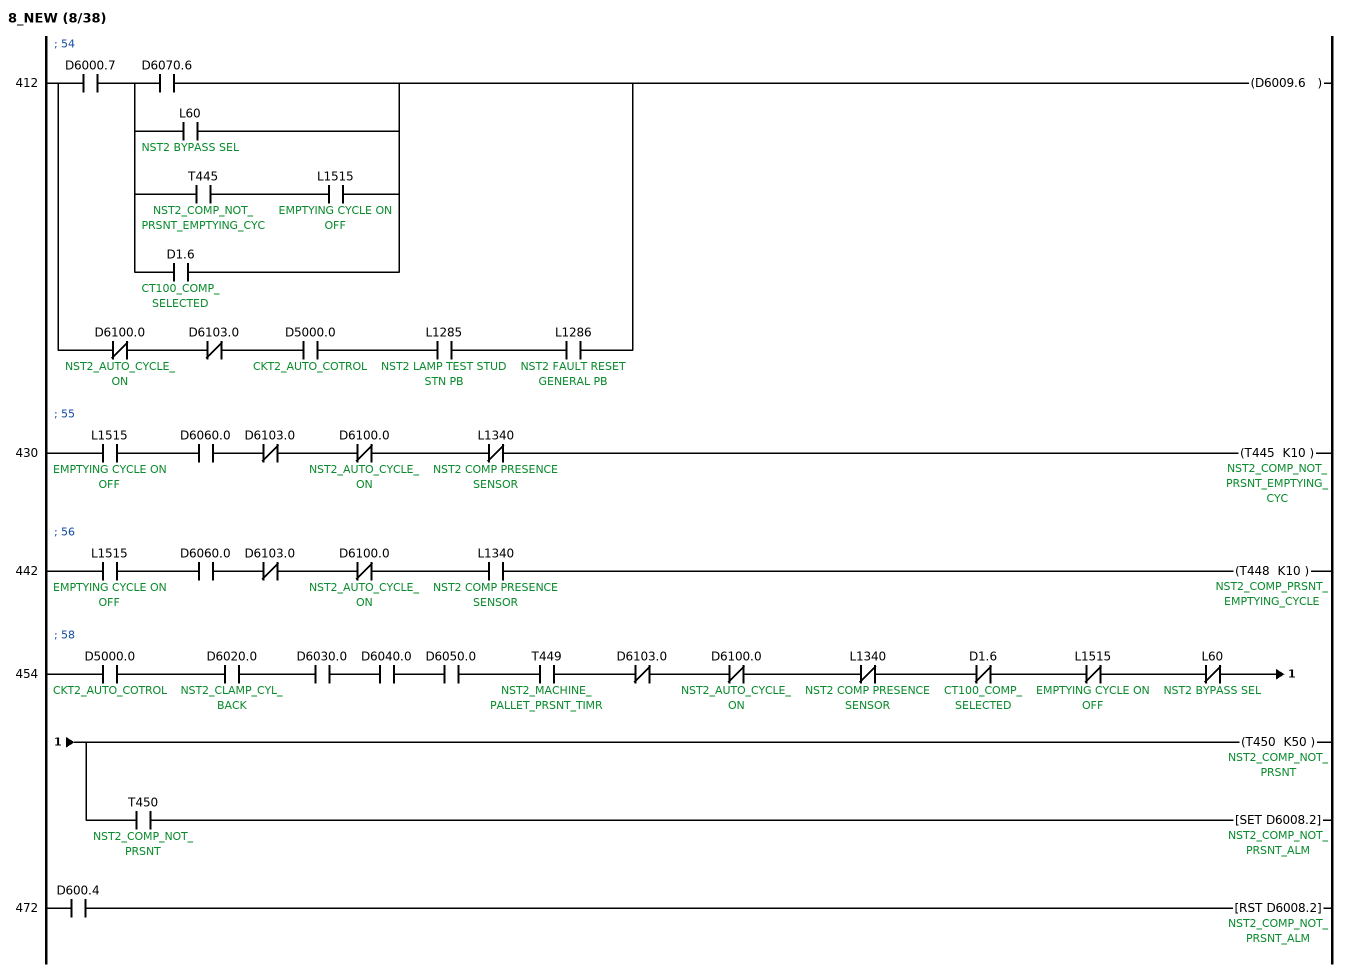
; 54
412   LD      D6000.7
      LD      D6070.6
      OR      L60  ; NST2 BYPASS SEL
      LD      T445  ; NST2_COMP_NOT_PRSNT_EMPTYING_CYC
      AND     L1515  ; EMPTYING CYCLE ON OFF
      ORB
      OR      D1.6  ; CT100_COMP_SELECTED
      ANB
      LDI     D6100.0  ; NST2_AUTO_CYCLE_ON
      ANI     D6103.0
      AND     D5000.0  ; CKT2_AUTO_COTROL
      AND     L1285  ; NST2 LAMP TEST STUD STN PB
      AND     L1286  ; NST2 FAULT RESET GENERAL PB
      ORB
      OUT     D6009.6
; 55
430   LD      L1515  ; EMPTYING CYCLE ON OFF
      AND     D6060.0
      ANI     D6103.0
      ANI     D6100.0  ; NST2_AUTO_CYCLE_ON
      ANI     L1340  ; NST2 COMP PRESENCE SENSOR
      OUT     T445 K10  ; NST2_COMP_NOT_PRSNT_EMPTYING_CYC
; 56
442   LD      L1515  ; EMPTYING CYCLE ON OFF
      AND     D6060.0
      ANI     D6103.0
      ANI     D6100.0  ; NST2_AUTO_CYCLE_ON
      AND     L1340  ; NST2 COMP PRESENCE SENSOR
      OUT     T448 K10  ; NST2_COMP_PRSNT_EMPTYING_CYCLE
; 58
454   LD      D5000.0  ; CKT2_AUTO_COTROL
      AND     D6020.0  ; NST2_CLAMP_CYL_BACK
      AND     D6030.0
      AND     D6040.0
      AND     D6050.0
      AND     T449  ; NST2_MACHINE_PALLET_PRSNT_TIMR
      ANI     D6103.0
      ANI     D6100.0  ; NST2_AUTO_CYCLE_ON
      ANI     L1340  ; NST2 COMP PRESENCE SENSOR
      ANI     D1.6  ; CT100_COMP_SELECTED
      ANI     L1515  ; EMPTYING CYCLE ON OFF
      ANI     L60  ; NST2 BYPASS SEL
      OUT     T450 K50  ; NST2_COMP_NOT_PRSNT
      AND     T450  ; NST2_COMP_NOT_PRSNT
      SET     D6008.2  ; NST2_COMP_NOT_PRSNT_ALM
472   LD      D600.4
      RST     D6008.2  ; NST2_COMP_NOT_PRSNT_ALM
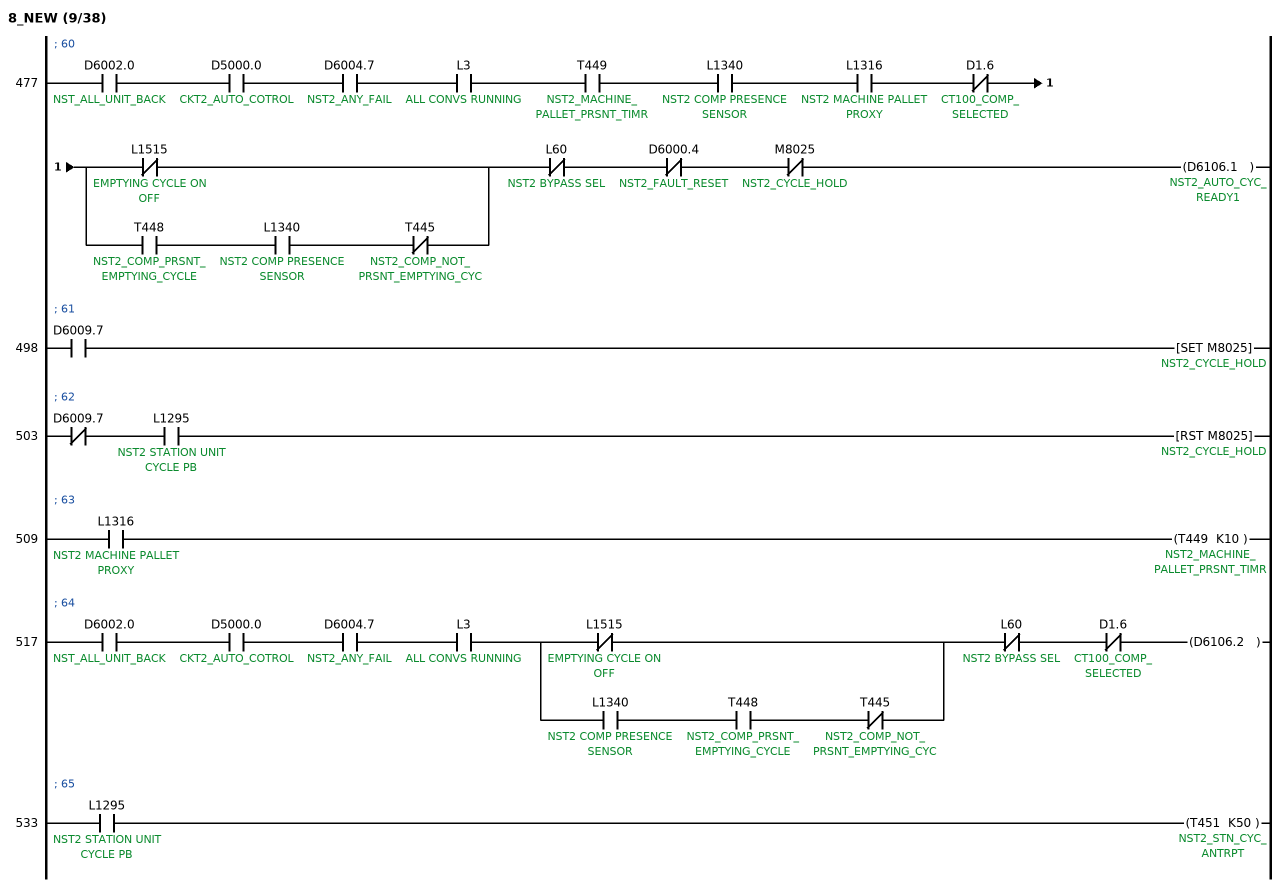
; 60
477   LD      D6002.0  ; NST_ALL_UNIT_BACK
      AND     D5000.0  ; CKT2_AUTO_COTROL
      AND     D6004.7  ; NST2_ANY_FAIL
      AND     L3  ; ALL CONVS RUNNING
      AND     T449  ; NST2_MACHINE_PALLET_PRSNT_TIMR
      AND     L1340  ; NST2 COMP PRESENCE SENSOR
      AND     L1316  ; NST2 MACHINE PALLET PROXY
      ANI     D1.6  ; CT100_COMP_SELECTED
      LDI     L1515  ; EMPTYING CYCLE ON OFF
      LD      T448  ; NST2_COMP_PRSNT_EMPTYING_CYCLE
      AND     L1340  ; NST2 COMP PRESENCE SENSOR
      ANI     T445  ; NST2_COMP_NOT_PRSNT_EMPTYING_CYC
      ORB
      ANB
      ANI     L60  ; NST2 BYPASS SEL
      ANI     D6000.4  ; NST2_FAULT_RESET
      ANI     M8025  ; NST2_CYCLE_HOLD
      OUT     D6106.1  ; NST2_AUTO_CYC_READY1
; 61
498   LD      D6009.7
      SET     M8025  ; NST2_CYCLE_HOLD
; 62
503   LDI     D6009.7
      AND     L1295  ; NST2 STATION UNIT CYCLE PB
      RST     M8025  ; NST2_CYCLE_HOLD
; 63
509   LD      L1316  ; NST2 MACHINE PALLET PROXY
      OUT     T449 K10  ; NST2_MACHINE_PALLET_PRSNT_TIMR
; 64
517   LD      D6002.0  ; NST_ALL_UNIT_BACK
      AND     D5000.0  ; CKT2_AUTO_COTROL
      AND     D6004.7  ; NST2_ANY_FAIL
      AND     L3  ; ALL CONVS RUNNING
      LDI     L1515  ; EMPTYING CYCLE ON OFF
      LD      L1340  ; NST2 COMP PRESENCE SENSOR
      AND     T448  ; NST2_COMP_PRSNT_EMPTYING_CYCLE
      ANI     T445  ; NST2_COMP_NOT_PRSNT_EMPTYING_CYC
      ORB
      ANB
      ANI     L60  ; NST2 BYPASS SEL
      ANI     D1.6  ; CT100_COMP_SELECTED
      OUT     D6106.2
; 65
533   LD      L1295  ; NST2 STATION UNIT CYCLE PB
      OUT     T451 K50  ; NST2_STN_CYC_ANTRPT
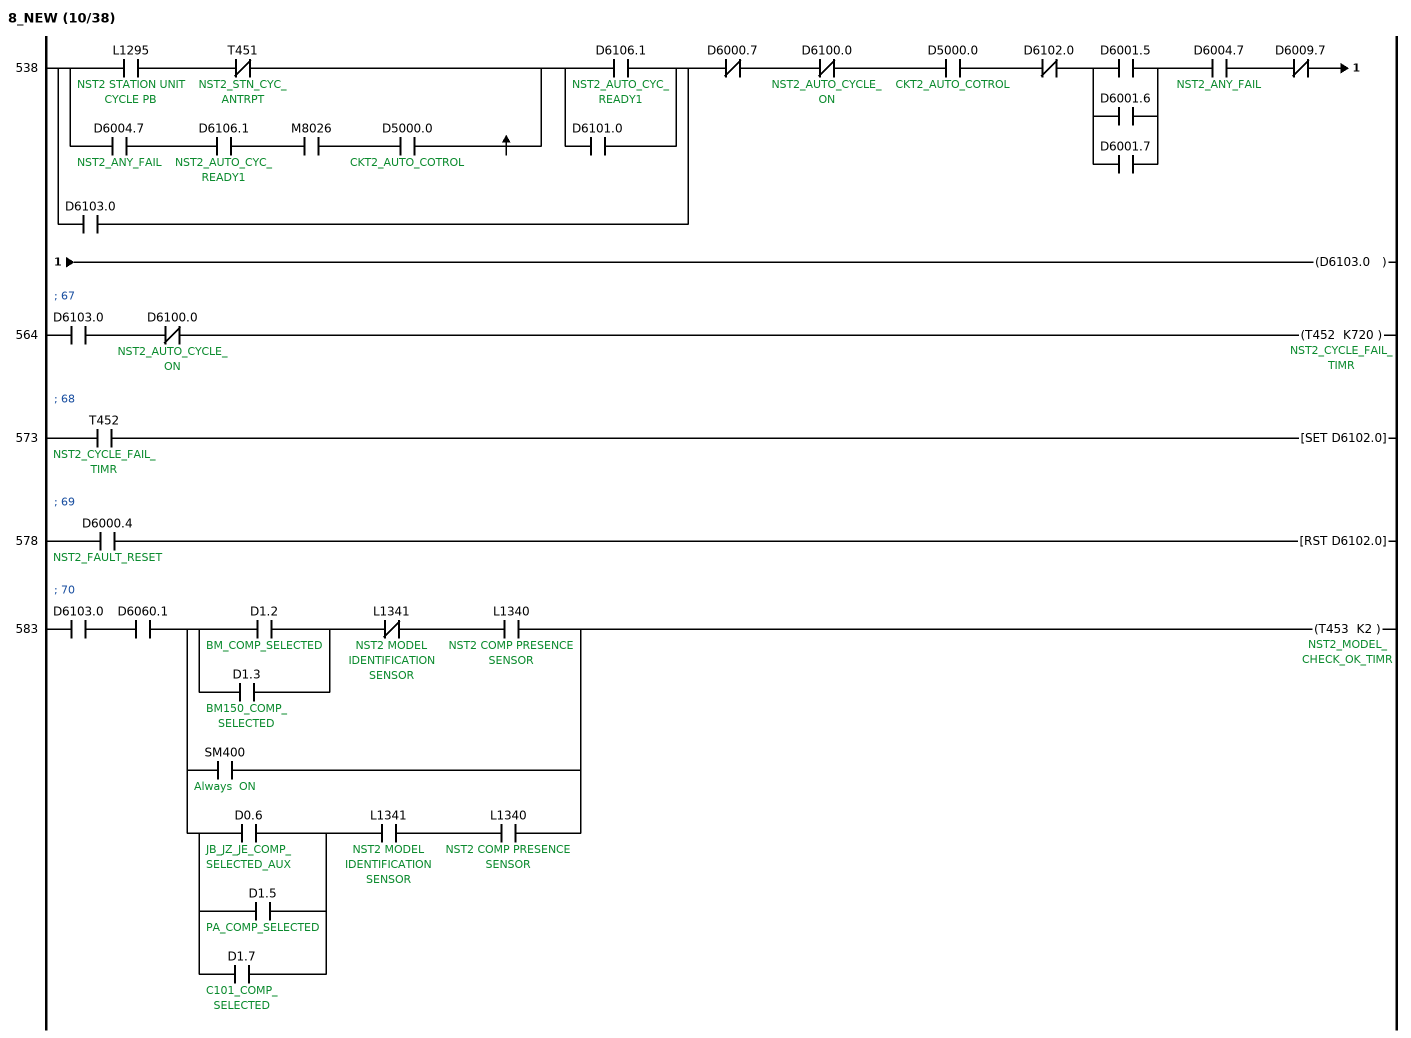
538   LD      L1295  ; NST2 STATION UNIT CYCLE PB
      ANI     T451  ; NST2_STN_CYC_ANTRPT
      LD      D6004.7  ; NST2_ANY_FAIL
      AND     D6106.1  ; NST2_AUTO_CYC_READY1
      AND     M8026
      AND     D5000.0  ; CKT2_AUTO_COTROL
      MEP
      ORB
      LD      D6106.1  ; NST2_AUTO_CYC_READY1
      OR      D6101.0
      ANB
      OR      D6103.0
      ANI     D6000.7
      ANI     D6100.0  ; NST2_AUTO_CYCLE_ON
      AND     D5000.0  ; CKT2_AUTO_COTROL
      ANI     D6102.0
      LD      D6001.5
      OR      D6001.6
      OR      D6001.7
      ANB
      AND     D6004.7  ; NST2_ANY_FAIL
      ANI     D6009.7
      OUT     D6103.0
; 67
564   LD      D6103.0
      ANI     D6100.0  ; NST2_AUTO_CYCLE_ON
      OUT     T452 K720  ; NST2_CYCLE_FAIL_TIMR
; 68
573   LD      T452  ; NST2_CYCLE_FAIL_TIMR
      SET     D6102.0
; 69
578   LD      D6000.4  ; NST2_FAULT_RESET
      RST     D6102.0
; 70
583   LD      D6103.0
      AND     D6060.1
      LD      D1.2  ; BM_COMP_SELECTED
      OR      D1.3  ; BM150_COMP_SELECTED
      ANI     L1341  ; NST2 MODEL IDENTIFICATION SENSOR
      AND     L1340  ; NST2 COMP PRESENCE SENSOR
      OR      SM400  ; Always  ON
      LD      D0.6  ; JB_JZ_JE_COMP_SELECTED_AUX
      OR      D1.5  ; PA_COMP_SELECTED
      OR      D1.7  ; C101_COMP_SELECTED
      AND     L1341  ; NST2 MODEL IDENTIFICATION SENSOR
      AND     L1340  ; NST2 COMP PRESENCE SENSOR
      ORB
      ANB
      OUT     T453 K2  ; NST2_MODEL_CHECK_OK_TIMR
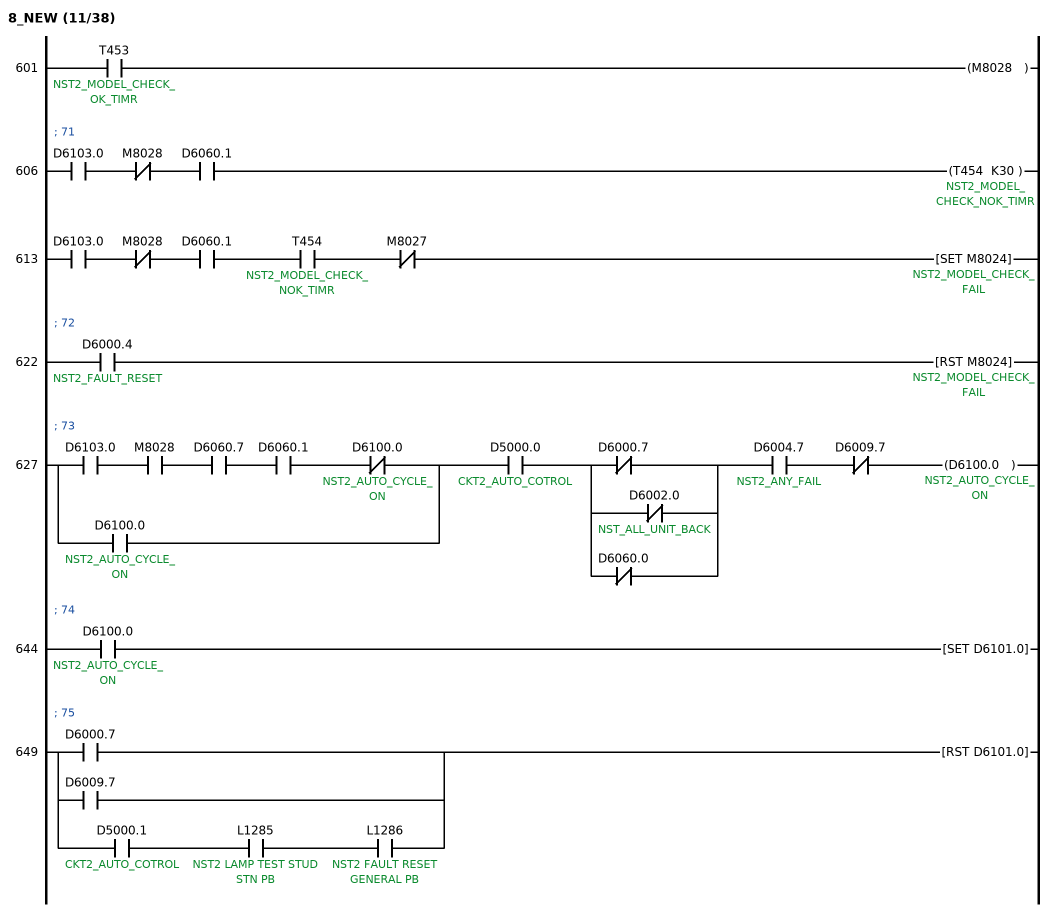
601   LD      T453  ; NST2_MODEL_CHECK_OK_TIMR
      OUT     M8028
; 71
606   LD      D6103.0
      ANI     M8028
      AND     D6060.1
      OUT     T454 K30  ; NST2_MODEL_CHECK_NOK_TIMR
613   LD      D6103.0
      ANI     M8028
      AND     D6060.1
      AND     T454  ; NST2_MODEL_CHECK_NOK_TIMR
      ANI     M8027
      SET     M8024  ; NST2_MODEL_CHECK_FAIL
; 72
622   LD      D6000.4  ; NST2_FAULT_RESET
      RST     M8024  ; NST2_MODEL_CHECK_FAIL
; 73
627   LD      D6103.0
      AND     M8028
      AND     D6060.7
      AND     D6060.1
      ANI     D6100.0  ; NST2_AUTO_CYCLE_ON
      OR      D6100.0  ; NST2_AUTO_CYCLE_ON
      AND     D5000.0  ; CKT2_AUTO_COTROL
      LDI     D6000.7
      ORI     D6002.0  ; NST_ALL_UNIT_BACK
      ORI     D6060.0
      ANB
      AND     D6004.7  ; NST2_ANY_FAIL
      ANI     D6009.7
      OUT     D6100.0  ; NST2_AUTO_CYCLE_ON
; 74
644   LD      D6100.0  ; NST2_AUTO_CYCLE_ON
      SET     D6101.0
; 75
649   LD      D6000.7
      OR      D6009.7
      LD      D5000.1  ; CKT2_AUTO_COTROL
      AND     L1285  ; NST2 LAMP TEST STUD STN PB
      AND     L1286  ; NST2 FAULT RESET GENERAL PB
      ORB
      RST     D6101.0
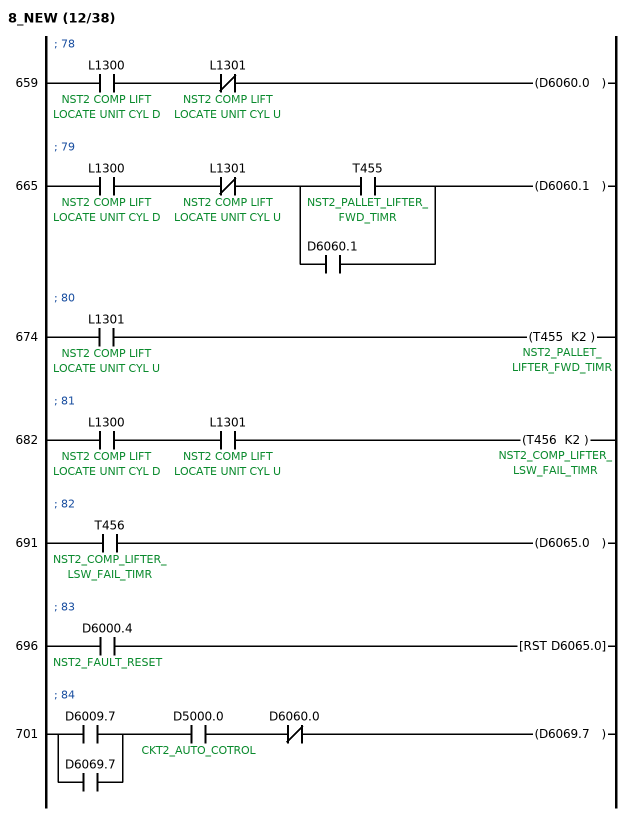
; 78
659   LD      L1300  ; NST2 COMP LIFT LOCATE UNIT CYL D
      ANI     L1301  ; NST2 COMP LIFT LOCATE UNIT CYL U
      OUT     D6060.0
; 79
665   LD      L1300  ; NST2 COMP LIFT LOCATE UNIT CYL D
      ANI     L1301  ; NST2 COMP LIFT LOCATE UNIT CYL U
      LD      T455  ; NST2_PALLET_LIFTER_FWD_TIMR
      OR      D6060.1
      ANB
      OUT     D6060.1
; 80
674   LD      L1301  ; NST2 COMP LIFT LOCATE UNIT CYL U
      OUT     T455 K2  ; NST2_PALLET_LIFTER_FWD_TIMR
; 81
682   LD      L1300  ; NST2 COMP LIFT LOCATE UNIT CYL D
      AND     L1301  ; NST2 COMP LIFT LOCATE UNIT CYL U
      OUT     T456 K2  ; NST2_COMP_LIFTER_LSW_FAIL_TIMR
; 82
691   LD      T456  ; NST2_COMP_LIFTER_LSW_FAIL_TIMR
      OUT     D6065.0
; 83
696   LD      D6000.4  ; NST2_FAULT_RESET
      RST     D6065.0
; 84
701   LD      D6009.7
      OR      D6069.7
      AND     D5000.0  ; CKT2_AUTO_COTROL
      ANI     D6060.0
      OUT     D6069.7
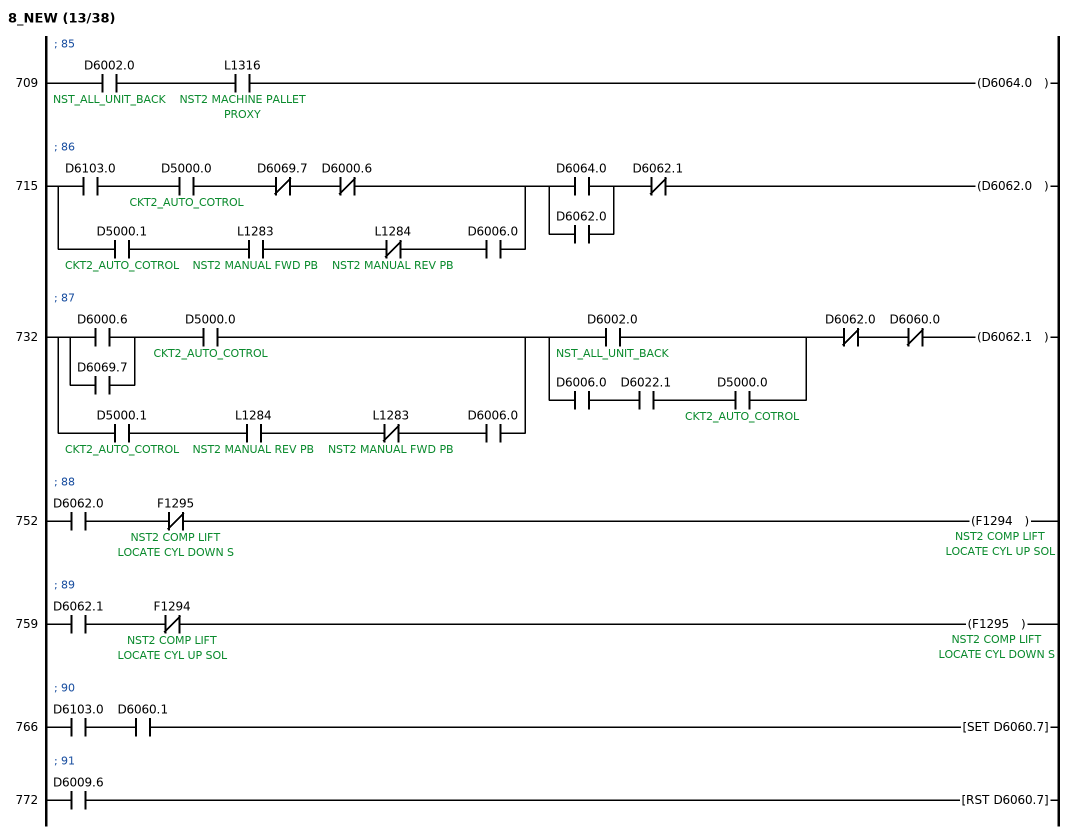
; 85
709   LD      D6002.0  ; NST_ALL_UNIT_BACK
      AND     L1316  ; NST2 MACHINE PALLET PROXY
      OUT     D6064.0
; 86
715   LD      D6103.0
      AND     D5000.0  ; CKT2_AUTO_COTROL
      ANI     D6069.7
      ANI     D6000.6
      LD      D5000.1  ; CKT2_AUTO_COTROL
      AND     L1283  ; NST2 MANUAL FWD PB
      ANI     L1284  ; NST2 MANUAL REV PB
      AND     D6006.0
      ORB
      LD      D6064.0
      OR      D6062.0
      ANB
      ANI     D6062.1
      OUT     D6062.0
; 87
732   LD      D6000.6
      OR      D6069.7
      AND     D5000.0  ; CKT2_AUTO_COTROL
      LD      D5000.1  ; CKT2_AUTO_COTROL
      AND     L1284  ; NST2 MANUAL REV PB
      ANI     L1283  ; NST2 MANUAL FWD PB
      AND     D6006.0
      ORB
      LD      D6002.0  ; NST_ALL_UNIT_BACK
      LD      D6006.0
      AND     D6022.1
      AND     D5000.0  ; CKT2_AUTO_COTROL
      ORB
      ANB
      ANI     D6062.0
      ANI     D6060.0
      OUT     D6062.1
; 88
752   LD      D6062.0
      ANI     F1295  ; NST2 COMP LIFT LOCATE CYL DOWN S
      OUT     F1294  ; NST2 COMP LIFT LOCATE CYL UP SOL
; 89
759   LD      D6062.1
      ANI     F1294  ; NST2 COMP LIFT LOCATE CYL UP SOL
      OUT     F1295  ; NST2 COMP LIFT LOCATE CYL DOWN S
; 90
766   LD      D6103.0
      AND     D6060.1
      SET     D6060.7
; 91
772   LD      D6009.6
      RST     D6060.7
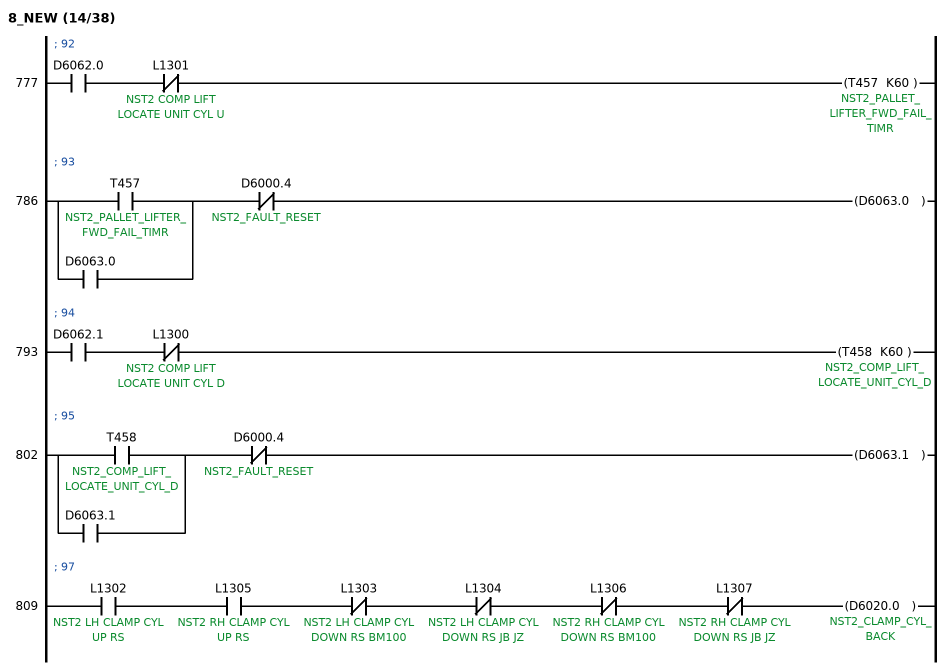
; 92
777   LD      D6062.0
      ANI     L1301  ; NST2 COMP LIFT LOCATE UNIT CYL U
      OUT     T457 K60  ; NST2_PALLET_LIFTER_FWD_FAIL_TIMR
; 93
786   LD      T457  ; NST2_PALLET_LIFTER_FWD_FAIL_TIMR
      OR      D6063.0
      ANI     D6000.4  ; NST2_FAULT_RESET
      OUT     D6063.0
; 94
793   LD      D6062.1
      ANI     L1300  ; NST2 COMP LIFT LOCATE UNIT CYL D
      OUT     T458 K60  ; NST2_COMP_LIFT_LOCATE_UNIT_CYL_D
; 95
802   LD      T458  ; NST2_COMP_LIFT_LOCATE_UNIT_CYL_D
      OR      D6063.1
      ANI     D6000.4  ; NST2_FAULT_RESET
      OUT     D6063.1
; 97
809   LD      L1302  ; NST2 LH CLAMP CYL UP RS
      AND     L1305  ; NST2 RH CLAMP CYL UP RS
      ANI     L1303  ; NST2 LH CLAMP CYL DOWN RS BM100
      ANI     L1304  ; NST2 LH CLAMP CYL DOWN RS JB JZ
      ANI     L1306  ; NST2 RH CLAMP CYL DOWN RS BM100
      ANI     L1307  ; NST2 RH CLAMP CYL DOWN RS JB JZ
      OUT     D6020.0  ; NST2_CLAMP_CYL_BACK
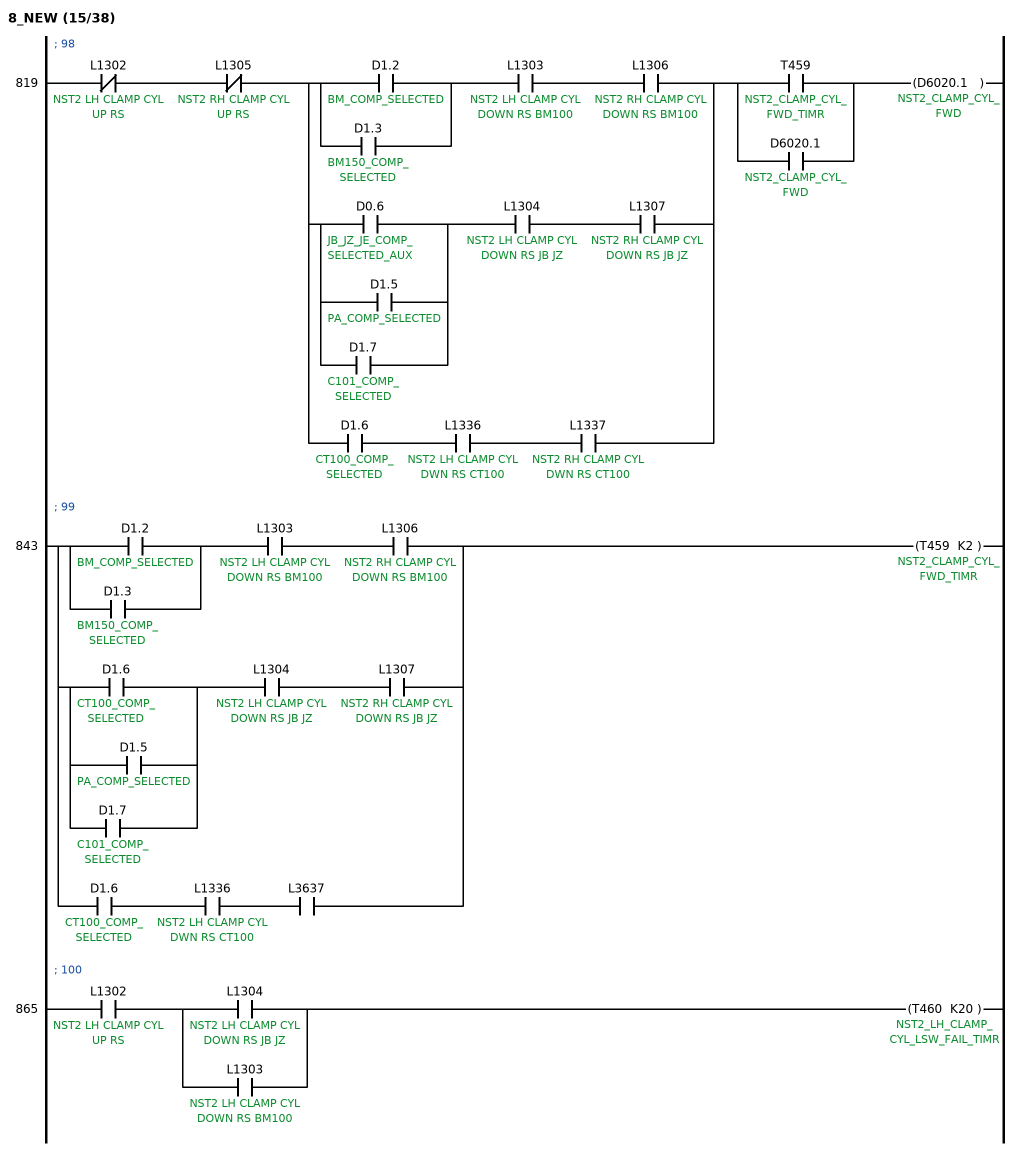
; 98
819   LDI     L1302  ; NST2 LH CLAMP CYL UP RS
      ANI     L1305  ; NST2 RH CLAMP CYL UP RS
      LD      D1.2  ; BM_COMP_SELECTED
      OR      D1.3  ; BM150_COMP_SELECTED
      AND     L1303  ; NST2 LH CLAMP CYL DOWN RS BM100
      AND     L1306  ; NST2 RH CLAMP CYL DOWN RS BM100
      LD      D0.6  ; JB_JZ_JE_COMP_SELECTED_AUX
      OR      D1.5  ; PA_COMP_SELECTED
      OR      D1.7  ; C101_COMP_SELECTED
      AND     L1304  ; NST2 LH CLAMP CYL DOWN RS JB JZ
      AND     L1307  ; NST2 RH CLAMP CYL DOWN RS JB JZ
      ORB
      LD      D1.6  ; CT100_COMP_SELECTED
      AND     L1336  ; NST2 LH CLAMP CYL DWN RS CT100
      AND     L1337  ; NST2 RH CLAMP CYL DWN RS CT100
      ORB
      ANB
      LD      T459  ; NST2_CLAMP_CYL_FWD_TIMR
      OR      D6020.1  ; NST2_CLAMP_CYL_FWD
      ANB
      OUT     D6020.1  ; NST2_CLAMP_CYL_FWD
; 99
843   LD      D1.2  ; BM_COMP_SELECTED
      OR      D1.3  ; BM150_COMP_SELECTED
      AND     L1303  ; NST2 LH CLAMP CYL DOWN RS BM100
      AND     L1306  ; NST2 RH CLAMP CYL DOWN RS BM100
      LD      D1.6  ; CT100_COMP_SELECTED
      OR      D1.5  ; PA_COMP_SELECTED
      OR      D1.7  ; C101_COMP_SELECTED
      AND     L1304  ; NST2 LH CLAMP CYL DOWN RS JB JZ
      AND     L1307  ; NST2 RH CLAMP CYL DOWN RS JB JZ
      ORB
      LD      D1.6  ; CT100_COMP_SELECTED
      AND     L1336  ; NST2 LH CLAMP CYL DWN RS CT100
      AND     L3637
      ORB
      OUT     T459 K2  ; NST2_CLAMP_CYL_FWD_TIMR
; 100
865   LD      L1302  ; NST2 LH CLAMP CYL UP RS
      LD      L1304  ; NST2 LH CLAMP CYL DOWN RS JB JZ
      OR      L1303  ; NST2 LH CLAMP CYL DOWN RS BM100
      ANB
      OUT     T460 K20  ; NST2_LH_CLAMP_CYL_LSW_FAIL_TIMR
